# B&R Automation Studio project TD52 (part 119)

#### Cyclic.st - Cyclic code
```iecst
(*******************************************************************************
Ansl configuration for the Plant Communication

This code is confidential and proprietary to the INNIO Company.
It may not be used in any form, or reproduced in any manner, without the express
written permission of the INNIO Company.
Copyright, INNIO Company, 2024

Customized modifications: -
------------------------

History:
-------
V4.14.0	26.11.2024	Astner	Created Task

Instructions for use:
--------------------
The Configuration of the ANSL Communication is executed automatically when valid Parameter Values are configured.
If the Communication to the Master Control is redundant, set the variable bRedundantMasterEnabled in the Init Task.

Outstandings:
------------

*******************************************************************************)

PROGRAM _CYCLIC

	(* Parameters and Configuration Status for customized module *)
	OUT_HA.bPlantComCfgOk 		:= MM2VIS.tPlantComm.bCfg_OK;
		(* Start ANSL Configuration when parameter is set *)
	IF (EDGEPOS(Para.tPlantComm.bActive)) THEN
		MM2VIS.tPlantComm.bCfg_Err := FALSE;
		MM2VIS.tPlantComm.bCfg_OK := FALSE;
		MM2VIS.tPlantComm.bCfg_Rst := FALSE;
		iSTEP := GET_MODULE_NR;
	(* Stop ANSL Communication when parameter is unset *)
	ELSIF (EDGENEG(Para.tPlantComm.bActive)) THEN
		iSTEP := STOP_ANSL_COM;
		(* Exit Programm if parameter is not set *)
	ELSIF (NOT Para.tPlantComm.bActive AND NOT bPlantCommStopInProgress) THEN
		RETURN;
	END_IF;

	CASE iSTEP OF
		DATAOBJ_ERROR:
			(* Set HMI Diagnostics Error *)
			MM2VIS.tPlantComm.bCfg_Err := TRUE;
			MM2VIS.tPlantComm.bCfg_OK := FALSE;
			MM2VIS.tPlantComm.bCfg_Rst := FALSE;
			RETURN;
		ANSL_ERROR:
			(* Set HMI Diagnostics Error *)
			MM2VIS.tPlantComm.bCfg_Err := TRUE;
			MM2VIS.tPlantComm.bCfg_OK := FALSE;
			MM2VIS.tPlantComm.bCfg_Rst := FALSE;
			RETURN;
		GET_MODULE_NR:
			(* Set Engine Number to 1 for WinMOD Simulation *)
			IF (OUT_HA.bSimWinMOD_Active) THEN
				iThisEngineNr := 1;
				itoa(iThisEngineNr, ADR(strThisEngineNr));
				(* Reset Error bits*)
				MM2VIS.tPlantComm.bCfg_Err := FALSE;
				MM2VIS.tPlantComm.bCfg_OK := FALSE;
				MM2VIS.tPlantComm.bCfg_Rst := FALSE;
				(* Go to the next step *)
				iSTEP := PREP_DATAOBJ;
				RETURN;
			END_IF;
			(* Use Engine Number from HMI *)
			IF (IN_HA.iModule >= 1 AND IN_HA.iModule <= 32) THEN
				iThisEngineNr := IN_HA.iModule;
				itoa(iThisEngineNr, ADR(strThisEngineNr));
			ELSE
				MM2VIS.tPlantComm.bCfg_Err := TRUE;
				MM2VIS.tPlantComm.bCfg_OK := FALSE;
				MM2VIS.tPlantComm.bCfg_Rst := FALSE;
				RETURN;
			END_IF;
			IF (Para.tPlantComm.iEng_Num_Min = 0 AND Para.tPlantComm.iEng_Num_Max = 0) THEN
				bEng2EngComEnabled := FALSE;
			ELSIF (Para.tPlantComm.iEng_Num_Min > Para.tPlantComm.iEng_Num_Max) THEN
				MM2VIS.tPlantComm.bCfg_Err := TRUE;
				MM2VIS.tPlantComm.bCfg_OK := FALSE;
				MM2VIS.tPlantComm.bCfg_Rst := FALSE;
				RETURN;
			(* Out of bounds check *)
			ELSIF (Para.tPlantComm.iEng_Num_Min < 1 OR Para.tPlantComm.iEng_Num_Min > 32 OR Para.tPlantComm.iEng_Num_Max < 1 OR Para.tPlantComm.iEng_Num_Max > 32) THEN
				MM2VIS.tPlantComm.bCfg_Err := TRUE;
				MM2VIS.tPlantComm.bCfg_OK := FALSE;
				MM2VIS.tPlantComm.bCfg_Rst := FALSE;
				RETURN;
			ELSE
				bEng2EngComEnabled := TRUE;
				iEngNumMin := Para.tPlantComm.iEng_Num_Min;
				iEngNumMax := Para.tPlantComm.iEng_Num_Max;
			END_IF;
			IF (Para.tPlantComm.iMas_Num_Min = 0 AND Para.tPlantComm.iMas_Num_Max = 0) THEN
				bEng2MasComEnabled := FALSE;
			ELSIF (Para.tPlantComm.iMas_Num_Min > Para.tPlantComm.iMas_Num_Max) THEN
				MM2VIS.tPlantComm.bCfg_Err := TRUE;
				MM2VIS.tPlantComm.bCfg_OK := FALSE;
				MM2VIS.tPlantComm.bCfg_Rst := FALSE;
				RETURN;
			ELSE
				bEng2MasComEnabled := TRUE;
				iMasNumMin := Para.tPlantComm.iMas_Num_Min;
				iMasNumMax := Para.tPlantComm.iMas_Num_Max;
			END_IF;

			(* Reset Error bits and continue with the next step *)
			MM2VIS.tPlantComm.bCfg_Err := FALSE;
			MM2VIS.tPlantComm.bCfg_OK := FALSE;
			MM2VIS.tPlantComm.bCfg_Rst := FALSE;
			iSTEP := PREP_DATAOBJ;

		PREP_DATAOBJ:
			(*** Creation of the ANSL Configuration Data Object ***)

			(* ANSL Header *)
			strcat(pANSL_config, ADR('<?xml version ="1.0" encoding="utf-8"?>'));
			strcat(pANSL_config, ADR('<AnslClient>'));
			strcat(pANSL_config, ADR('<Diag TimeStamp="HalIO::tDiagClient.TimeStamp" ClientConn="HalIO::tDiagClient.Conn" ClientConnErr="HalIO::tDiagClient.ConnErr"/>'));

			(********************************************************************)
			(*																	*)
			(*                   Communication to Master						*)
			(*																	*)
			(********************************************************************)

			IF (bEng2MasComEnabled) THEN
				IF (NOT bRedundantMasterEnabled) THEN
					(* Add configured Masters to communication *)
					FOR x:=iMasNumMin TO iMasNumMax DO
						(* Check length of config object *)
						IF strlen(pANSL_config) > iANSL_config_length_max - 1000 THEN
							iSTEP := DATAOBJ_ERROR;
							RETURN;
						END_IF;
						(* Convert current asset numbers to strings *)
						strCurrentAssetNum 	:= '';
						strCurrentAssetSub 	:= '';
						strCurrentAssetIP 	:= '';
						itoa(x, ADR(strCurrentAssetNum));
						itoa(iMastersSUB[x], ADR(strCurrentAssetSub));
						itoa(iMastersIP[x], ADR(strCurrentAssetIP));

						//Line 1
						strcat(pANSL_config, ADR('<Connection ConnName="Master'));
						strcat(pANSL_config, ADR(strCurrentAssetNum));
						strcat(pANSL_config, ADR('" TargetAddr="192.168.'));
						strcat(pANSL_config, ADR(strCurrentAssetSub));
						strcat(pANSL_config, ADR('.'));
						strcat(pANSL_config, ADR(strCurrentAssetIP));
						strcat(pANSL_config, ADR('" AnslPort="11179" Timeout="5000" SendDelay="2" BfSize="65536" ConnMode="0" EnableSSL="1" SSLConfig="SSL_Eng'));
						strcat(pANSL_config, ADR(strThisEngineNr));
						strcat(pANSL_config, ADR('" PW="'));
						strcat(pANSL_config, ADR(strAnsl_Com_Pw));
						strcat(pANSL_config, ADR('">'));
						// Line 2
						strcat(pANSL_config, ADR('<Diag ConnErr="HalIO::tDiagMaster['));
						strcat(pANSL_config, ADR(strCurrentAssetNum));
						strcat(pANSL_config, ADR('].Err" ConnPvWrite="HalIO::tDiagMaster['));
						strcat(pANSL_config, ADR(strCurrentAssetNum));
						strcat(pANSL_config, ADR('].PvWrite" ConnPvWriteErr="HalIO::tDiagMaster['));
						strcat(pANSL_config, ADR(strCurrentAssetNum));
						strcat(pANSL_config, ADR('].PvWriteErr" ConnPvReadErr="HalIO::tDiagMaster['));
						strcat(pANSL_config, ADR(strCurrentAssetNum));
						strcat(pANSL_config, ADR('].PvReadErr"/>'));
						// Line 3
						strcat(pANSL_config, ADR('<PVS>'));
						// Line 4
						strcat(pANSL_config, ADR('<Read LocalPvName="HalIO::tPlantCom_M2E_In_100ms['));
						strcat(pANSL_config, ADR(strCurrentAssetNum));
						strcat(pANSL_config, ADR(']" RemotePvName="HalIO::tPlantCom_M2E_Out_100ms['));
						strcat(pANSL_config, ADR(strThisEngineNr));
						strcat(pANSL_config, ADR(']" DefaultValue="0" SyncPv="0" RefreshRate="100" Hysteresis="0"/>'));
						// Line 5
						strcat(pANSL_config, ADR('<Read LocalPvName="HalIO::tPlantCom_M2E_In_10ms['));
						strcat(pANSL_config, ADR(strCurrentAssetNum));
						strcat(pANSL_config, ADR(']" RemotePvName="HalIO::tPlantCom_M2E_Out_10ms['));
						strcat(pANSL_config, ADR(strThisEngineNr));
						strcat(pANSL_config, ADR(']" DefaultValue="0" SyncPv="0" RefreshRate="10" Hysteresis="0"/>'));
						// Line 6
						strcat(pANSL_config, ADR('</PVS>'));
						// Line 7
						strcat(pANSL_config, ADR('</Connection>'));
					END_FOR
				ELSE
					(********************************************************************)
					(*																	*)
					(*                 Communication to Redundant Master				*)
					(*																	*)
					(********************************************************************)

					(* Check length of config object *)
					IF strlen(pANSL_config) > iANSL_config_length_max - 1000 THEN
						iSTEP := DATAOBJ_ERROR;
						RETURN;
					END_IF;
					(* Convert current asset numbers to strings *)
					strCurrentAssetNum 	:= '';
					strCurrentAssetSub 	:= '';
					strCurrentAssetIP 	:= '';
					itoa(1, ADR(strCurrentAssetNum));
					itoa(iMastersSUB[1], ADR(strCurrentAssetSub));
					itoa(iMastersIP[1], ADR(strCurrentAssetIP));

					//Line 1
					strcat(pANSL_config, ADR('<Connection ConnName="Master'));
					strcat(pANSL_config, ADR(strCurrentAssetNum));
					strcat(pANSL_config, ADR('" TargetAddr="192.168.'));
					strcat(pANSL_config, ADR(strCurrentAssetSub));
					strcat(pANSL_config, ADR('.'));
					strcat(pANSL_config, ADR(strCurrentAssetIP));
					strcat(pANSL_config, ADR('" AnslPort="11169" Timeout="5000" SendDelay="2" BfSize="65536" ConnMode="1" EnableSSL="0" SSLConfig="SSL_Eng'));
					strcat(pANSL_config, ADR(strThisEngineNr));
					strcat(pANSL_config, ADR('" PW="'));
					strcat(pANSL_config, ADR(strAnsl_Com_Pw));
					strcat(pANSL_config, ADR('">'));
					// Line 2
					strcat(pANSL_config, ADR('<Diag ConnErr="HalIO::tDiagMaster['));
					strcat(pANSL_config, ADR(strCurrentAssetNum));
					strcat(pANSL_config, ADR('].Err" ConnPvWrite="HalIO::tDiagMaster['));
					strcat(pANSL_config, ADR(strCurrentAssetNum));
					strcat(pANSL_config, ADR('].PvWrite" ConnPvWriteErr="HalIO::tDiagMaster['));
					strcat(pANSL_config, ADR(strCurrentAssetNum));
					strcat(pANSL_config, ADR('].PvWriteErr" ConnPvReadErr="HalIO::tDiagMaster['));
					strcat(pANSL_config, ADR(strCurrentAssetNum));
					strcat(pANSL_config, ADR('].PvReadErr" RedConnActIpAddr="HalIO::tDiagMaster['));
					strcat(pANSL_config, ADR(strCurrentAssetNum));
					strcat(pANSL_config, ADR('].RedConnActIpAddr" RedConnAct="HalIO::tDiagMaster['));
					strcat(pANSL_config, ADR(strCurrentAssetNum));
					strcat(pANSL_config, ADR('].RedConnAct" RedConnState="HalIO::tDiagMaster['));
					strcat(pANSL_config, ADR(strCurrentAssetNum));
					strcat(pANSL_config, ADR('].RedConnState"/>'));
					// Line 3
					strcat(pANSL_config, ADR('<PVS>'));
					// Line 4
					strcat(pANSL_config, ADR('<Read LocalPvName="HalIO::tPlantCom_M2E_In_100ms['));
					strcat(pANSL_config, ADR(strCurrentAssetNum));
					strcat(pANSL_config, ADR(']" RemotePvName="HalIO::tPlantCom_M2E_Out_100ms['));
					strcat(pANSL_config, ADR(strThisEngineNr));
					strcat(pANSL_config, ADR(']" DefaultValue="0" SyncPv="0" RefreshRate="100" Hysteresis="0"/>'));
					// Line 5
					strcat(pANSL_config, ADR('<Read LocalPvName="HalIO::tPlantCom_M2E_In_10ms['));
					strcat(pANSL_config, ADR(strCurrentAssetNum));
					strcat(pANSL_config, ADR(']" RemotePvName="HalIO::tPlantCom_M2E_Out_10ms['));
					strcat(pANSL_config, ADR(strThisEngineNr));
					strcat(pANSL_config, ADR(']" DefaultValue="0" SyncPv="0" RefreshRate="10" Hysteresis="0"/>'));
					// Line 6
					strcat(pANSL_config, ADR('</PVS>'));
					// Line 7
					strcat(pANSL_config, ADR('</Connection>'));
				END_IF
			END_IF

			(********************************************************************)
			(*																	*)
			(*                   Communication to Engines						*)
			(*																	*)
			(********************************************************************)

			IF (bEng2EngComEnabled) THEN
				(* Add configured Engines to communication *)
				FOR x:=iEngNumMin TO iEngNumMax DO
					(* Check length of config object *)
					IF strlen(pANSL_config) > iANSL_config_length_max - 1000 THEN
						iSTEP := DATAOBJ_ERROR;
						RETURN;
					END_IF;

					IF (x <> iThisEngineNr) THEN
						(* Convert current asset numbers to strings *)
						strCurrentAssetNum 	:= '';
						strCurrentAssetSub 	:= '';
						strCurrentAssetIP 	:= '';
						itoa(x, ADR(strCurrentAssetNum));
						itoa(iEnginesSUB[x], ADR(strCurrentAssetSub));
						itoa(iEnginesIP[x], ADR(strCurrentAssetIP));

						//Line 1
						strcat(pANSL_config, ADR('<Connection ConnName="Engine'));
						strcat(pANSL_config, ADR(strCurrentAssetNum));
						strcat(pANSL_config, ADR('" TargetAddr="192.168.'));
						strcat(pANSL_config, ADR(strCurrentAssetSub));
						strcat(pANSL_config, ADR('.'));
						strcat(pANSL_config, ADR(strCurrentAssetIP));
						strcat(pANSL_config, ADR('" AnslPort="11179" Timeout="5000" SendDelay="2" BfSize="65536" ConnMode="0" EnableSSL="1" SSLConfig="SSL_Eng'));
						strcat(pANSL_config, ADR(strThisEngineNr));
						strcat(pANSL_config, ADR('"> PW="'));
						strcat(pANSL_config, ADR(strAnsl_Com_Pw));
						strcat(pANSL_config, ADR('"'));

						// Line 2
						strcat(pANSL_config, ADR('<Diag ConnErr="HalIO::tDiagEngine['));
						strcat(pANSL_config, ADR(strCurrentAssetNum));
						strcat(pANSL_config, ADR('].Err" ConnPvWrite="HalIO::tDiagEngine['));
						strcat(pANSL_config, ADR(strCurrentAssetNum));
						strcat(pANSL_config, ADR('].PvWrite" ConnPvWriteErr="HalIO::tDiagEngine['));
						strcat(pANSL_config, ADR(strCurrentAssetNum));
						strcat(pANSL_config, ADR('].PvWriteErr" ConnPvReadErr="HalIO::tDiagEngine['));
						strcat(pANSL_config, ADR(strCurrentAssetNum));
						strcat(pANSL_config, ADR('].PvReadErr"/>'));
						// Line 3
						strcat(pANSL_config, ADR('<PVS>'));
						// Line 4
						strcat(pANSL_config, ADR('<Read LocalPvName="HalIO::tPlantCom_E2E_In_100ms['));
						strcat(pANSL_config, ADR(strCurrentAssetNum));
						strcat(pANSL_config, ADR(']" RemotePvName="HalIO::tPlantCom_E2E_Out_100ms" DefaultValue="0" SyncPv="0" RefreshRate="100" Hysteresis="0"/>'));
						// Line 5
						strcat(pANSL_config, ADR('<Read LocalPvName="HalIO::tPlantCom_E2E_In_10ms['));
						strcat(pANSL_config, ADR(strCurrentAssetNum));
						strcat(pANSL_config, ADR(']" RemotePvName="HalIO::tPlantCom_E2E_Out_10ms" DefaultValue="0" SyncPv="0" RefreshRate="10" Hysteresis="0"/>'));
						// Line 6
						strcat(pANSL_config, ADR('</PVS>'));
						// Line 7
						strcat(pANSL_config, ADR('</Connection>'));
					END_IF
				END_FOR
			END_IF

			(* ANSL Footer*)
			strcat(pANSL_config, ADR('</AnslClient>'));

			(* Reset Error bits and continue with the next step *)
			MM2VIS.tPlantComm.bCfg_Err 				:= FALSE;
			MM2VIS.tPlantComm.bCfg_OK 				:= FALSE;
			MM2VIS.tPlantComm.bCfg_Rst 				:= FALSE;
			iSTEP := PREP_CHECK_DATAOBJ_STATUS;
		PREP_CHECK_DATAOBJ_STATUS:
			(* Prepare DataObjInfo Function Block *)
			xDatObjInfo_Ansl_Cfg.enable 			:= TRUE;
			xDatObjInfo_Ansl_Cfg.pName 				:= ADR(strAnslDataObjName);
			iSTEP := CHECK_DATAOBJ_STATUS;
		CHECK_DATAOBJ_STATUS:
			(* Check if DataObj already exists or has another error *)
			xDatObjInfo_Ansl_Cfg();
			(* Data object already exists *)
			IF (xDatObjInfo_Ansl_Cfg.status = ERR_OK) THEN
				xDatObjDelete_Ansl_Cfg.enable 		:= TRUE;
				xDatObjDelete_Ansl_Cfg.ident 		:= xDatObjInfo_Ansl_Cfg.ident;
				iSTEP := DELETE_DATAOBJ;
			ELSIF (xDatObjInfo_Ansl_Cfg.status = doERR_MODULNOTFOUND) THEN
				xDatObjCreate_Ansl_Cfg.enable 		:= TRUE;
				xDatObjCreate_Ansl_Cfg.pName 		:= ADR(strAnslDataObjName);
				xDatObjCreate_Ansl_Cfg.pCpyData 	:= pANSL_config;
				xDatObjCreate_Ansl_Cfg.MemType 		:= doUSRROM;
				xDatObjCreate_Ansl_Cfg.len 			:= strlen(pANSL_config);
				iSTEP 								:= CREATE_DATAOBJ;
			ELSIF (xDatObjInfo_Ansl_Cfg.status <> ERR_FUB_BUSY) THEN
				iSTEP 							:= DATAOBJ_ERROR;
			END_IF;
		DELETE_DATAOBJ:
			(* Delete Dataobj *)
			xDatObjDelete_Ansl_Cfg();
			IF (xDatObjDelete_Ansl_Cfg.status = ERR_OK) THEN
				xDatObjCreate_Ansl_Cfg.enable		:= TRUE;
				iSTEP 								:= CREATE_DATAOBJ;
			ELSIF (xDatObjDelete_Ansl_Cfg.status <> ERR_FUB_BUSY) THEN
				iSTEP						 		:= DATAOBJ_ERROR;
			END_IF;
		CREATE_DATAOBJ:
			IF (xDatObjCreate_Ansl_Cfg.len = 0) THEN
				iSTEP := PREP_DATAOBJ;
				RETURN;
			END_IF
			xDatObjCreate_Ansl_Cfg();
			IF (xDatObjCreate_Ansl_Cfg.status = ERR_OK) THEN
				strANSL_config 					:= '';
				xANSLClientStart.enable 		:= TRUE;
				xANSLClientStart.dataObjName 	:= strAnslDataObjName;
				iSTEP 							:= START_ANSL_COM;
			ELSIF (xDatObjCreate_Ansl_Cfg.status <> ERR_FUB_BUSY) THEN
				iSTEP						 	:= DATAOBJ_ERROR;
			END_IF;
		START_ANSL_COM:
			(* Only start ANSL Communication after all Software modules are loaded and running *)
			xANSLClientStart();
			IF (xANSLClientStart.status = ERR_OK) THEN
				xDatObjCreate_Ansl_Cfg.enable := FALSE;
				xDatObjDelete_Ansl_Cfg.enable := FALSE;
				xDatObjInfo_Ansl_Cfg.enable 	:= FALSE;
				MM2VIS.tPlantComm.bCfg_OK 	:= TRUE;
				iSTEP := PREP_ANSL_DIAGNOSTICS;
			ELSIF (xANSLClientStart.status <> ERR_FUB_BUSY) THEN
				iSTEP 						:= ANSL_ERROR;
			END_IF
		STOP_ANSL_COM:
			// todo test behaviour
			bPlantCommStopInProgress 			:= TRUE;
			xANSLClientStop.enable 				:= TRUE;
			xANSLClientStop.dataObjName 		:= strAnslDataObjName;
			xANSLClientStop();
			IF (xANSLClientStop.status = ERR_OK OR xANSLClientStop.status = asANSL_ERR_CLIENT_NOT_EXIST) THEN
				MM2VIS.tPlantComm.bCfg_OK 		:= FALSE;
				bPlantCommStopInProgress 		:= FALSE;
				(* Reset FUBs *)
				xANSLClientStart.dataObjName 	:= '';
				xANSLClientStart.enable			:= FALSE;
				xDatObjCreate_Ansl_Cfg.enable	:= FALSE;
				xDatObjCreate_Ansl_Cfg.len		:= 0;
				xDatObjCreate_Ansl_Cfg.pCpyData	:= 0;
				xDatObjInfo_Ansl_Cfg.enable		:= FALSE;
				xDatObjInfo_Ansl_Cfg.pName		:= 0;
				xDatObjDelete_Ansl_Cfg.enable	:= FALSE;
				xDatObjDelete_Ansl_Cfg.ident	:= 0;
				iSTEP := GET_MODULE_NR;
			ELSIF (xANSLClientStop.status <> ERR_FUB_BUSY) THEN
				iSTEP 							:= ANSL_ERROR;
			END_IF;
		PREP_ANSL_DIAGNOSTICS:
			iSTEP := ANSL_DIAGNOSTICS;
		ANSL_DIAGNOSTICS:
			(* Check for configuration changes *)
			IF (iEngNumMin <> Para.tPlantComm.iEng_Num_Min OR
				iEngNumMax <> Para.tPlantComm.iEng_Num_Max OR
				iMasNumMin <> Para.tPlantComm.iMas_Num_Min OR
				iMasNumMax <> Para.tPlantComm.iMas_Num_Max) THEN
				iSTEP := STOP_ANSL_COM;
			END_IF
			(* Evaluate Masters *)
			iNum_InterruptedMasters := 0;
			FOR x:=iMasNumMin TO iMasNumMax DO
				MM2VIS.tPlantComm.bMas_Ena[x] := tDiagMaster[x].Err = 0 AND tDiagMaster[x].PvReadErr = 0;
				IF (tDiagMaster[x].Err <> 0 OR tDiagMaster[x].PvReadErr <> 0) THEN
					iNum_InterruptedMasters := iNum_InterruptedMasters + 1;
				END_IF
			END_FOR

			(* Evaluate Engines *)
			iNum_InterruptedEngines := 0;
			FOR x:=iEngNumMin TO iEngNumMax DO
				IF (x = iThisEngineNr) THEN
					MM2VIS.tPlantComm.bEng_Ena[x] := TRUE;
				ELSE
					MM2VIS.tPlantComm.bEng_Ena[x] := tDiagEngine[x].Err = 0 AND tDiagEngine[x].PvReadErr = 0 AND x <> iThisEngineNr;
					IF (tDiagEngine[x].Err <> 0 OR tDiagEngine[x].PvReadErr <> 0) THEN
						iNum_InterruptedEngines := iNum_InterruptedEngines + 1;
					END_IF
				END_IF
			END_FOR

			(* Set warning variable *)
			bPlantComm_interrupted := iNum_InterruptedEngines <> 0 OR iNum_InterruptedMasters <> 0;

			(* Set/Unset GoodQual Values on connection interuptions/establishment *)
			FOR x:= iEngNumMin TO iEngNumMax DO
				IF (EDGENEG(MM2VIS.tPlantComm.bEng_Ena[x])) THEN
					FOR idx:=0 TO iDigArrayMax100ms DO
						tPlantCom_E2E_In_100ms[x].digitalSignals[idx].GoodQual := FALSE;
					END_FOR
					FOR idx:=0 TO iDigArrayMax10ms DO
						tPlantCom_E2E_In_10ms[x].digitalSignals[idx].GoodQual := FALSE;
					END_FOR
					FOR idx:=0 TO iAnaArrayMax100ms DO
						tPlantCom_E2E_In_100ms[x].analogSignals[idx].GoodQual := FALSE;
					END_FOR
					FOR idx:=0 TO iAnaArrayMax10ms DO
						tPlantCom_E2E_In_10ms[x].analogSignals[idx].GoodQual := FALSE;
					END_FOR
				END_IF
			END_FOR
			FOR x:= iMasNumMin TO iMasNumMax DO
				IF (EDGENEG(MM2VIS.tPlantComm.bMas_Ena[x])) THEN
					FOR idx:=0 TO iDigArrayMax100ms DO
						tPlantCom_M2E_In_100ms[x].digitalSignals[idx].GoodQual := FALSE;
					END_FOR
					FOR idx:=0 TO iDigArrayMax10ms DO
						tPlantCom_M2E_In_10ms[x].digitalSignals[idx].GoodQual := FALSE;
					END_FOR
					FOR idx:=0 TO iAnaArrayMax100ms DO
						tPlantCom_M2E_In_100ms[x].analogSignals[idx].GoodQual := FALSE;
					END_FOR
					FOR idx:=0 TO iAnaArrayMax10ms DO
						tPlantCom_M2E_In_10ms[x].analogSignals[idx].GoodQual := FALSE;
					END_FOR
				END_IF
			END_FOR
	END_CASE
END_PROGRAM
```

#### Init.st - Init code
```iecst
(*******************************************************************************
Ansl configuration for the Plant Communication

This code is confidential and proprietary to the INNIO Company.
It may not be used in any form, or reproduced in any manner, without the express
written permission of the INNIO Company.
Copyright, INNIO Company, 2024

Customized modifications: -
------------------------

History:
-------
V4.14.0	26.11.2024	Astner	Created Task

Instructions for use:
--------------------
The Configuration of the ANSL Communication is executed automatically when valid Parameter Values are configured.
If the Communication to the Master Control is redundant, set the variable bRedundantMasterEnabled in the Init Task.

Outstandings:
------------

*******************************************************************************)

PROGRAM _INIT
	(* Master 1 is redundant *)
	bRedundantMasterEnabled := FALSE;

	(* Default diagnostic bits *)
	MM2VIS.tPlantComm.bCfg_Err := FALSE;
	MM2VIS.tPlantComm.bCfg_OK  := FALSE;
	MM2VIS.tPlantComm.bCfg_Rst := FALSE;

	(* IP & SUBNET Masks *)
	FOR x:=1 TO 4 DO
		iMastersSUB[x]	:=	122;
		iMastersIP[x] 	:= 	30 + x;
	END_FOR

	FOR x:=1 TO 32 DO
		iEnginesSUB[x]	:=	122;
		iEnginesIP[x] 	:= 	10 + x;
	END_FOR
	(* Initialize Configuration Strings and Pointers *)
	strAnslDataObjName := 'HalIO::ANSLCom';
	strThisEngineNr := '';
	strCurrentAssetIP := '';
	strCurrentAssetSub := '';
	strCurrentAssetNum := '';
	strANSL_config := '';
	pANSL_config := ADR(strANSL_config);
	strAnsl_Com_Pw := 'vvsZKl2WtfuUhIlKaiANBLBnqHMr7jLXo7MDs/K0/P5wtUylYnR+0YUUjcfS9T0G';

	iSTEP := GET_MODULE_NR;

	tDiagClient;
	tDiagMaster;
	tDiagEngine;

END_PROGRAM
```

#### Variables.var - Local variables
```iecst
(*Configuration Step Variables*)
VAR
	iSTEP : USINT := 0;
END_VAR
VAR CONSTANT
	DATAOBJ_ERROR : USINT := 0;
	ANSL_ERROR : USINT := 1;
	GET_MODULE_NR : USINT := 2;
	PREP_DATAOBJ : USINT := 3;
	PREP_CHECK_DATAOBJ_STATUS : USINT := 4;
	CHECK_DATAOBJ_STATUS : USINT := 5;
	DELETE_DATAOBJ : USINT := 6;
	CREATE_DATAOBJ : USINT := 7;
	START_ANSL_COM : USINT := 8;
	STOP_ANSL_COM : USINT := 9;
	PREP_ANSL_DIAGNOSTICS : USINT := 10;
	ANSL_DIAGNOSTICS : USINT := 11;
END_VAR
VAR
	bPlantCommStopInProgress : BOOL := FALSE;
END_VAR
(*ANSL Config Variables*)
VAR
	strAnsl_Com_Pw : STRING[64] := ''; (*Password Hash for the encrypted ANSL Communication*)
	iThisEngineNr : USINT := 0; (*Engine number of this Engine*)
	strThisEngineNr : STRING[16] := ''; (*Engine number of this Engine*)
	iMastersSUB : ARRAY[0..4] OF USINT; (*Subnet Part of the IP of each master*)
	iMastersIP : ARRAY[0..4] OF USINT; (*Host Part of the IP of each master*)
	iEnginesSUB : ARRAY[0..32] OF USINT; (*Subnet Part of the IP of each engine*)
	iEnginesIP : ARRAY[0..32] OF USINT; (*Host Part of the IP of each engine*)
	idx : USINT := 0; (*loop iterator used to iterate over signals*)
	x : USINT := 0; (*loop iterator used to iterate over the communication participants*)
END_VAR
VAR CONSTANT
	iANSL_config_length_max : UINT := 60000; (*max dataobject length*)
END_VAR
VAR
	strANSL_config : STRING[iANSL_config_length_max] := ''; (*Ansl configuration string*)
	pANSL_config : UDINT := 0; (*Pointer to the Ansl configuration string*)
	strCurrentAssetNum : STRING[16] := ''; (*Strings of the dynamic values that are used to build the ansl dataoject*)
	strCurrentAssetSub : STRING[16] := ''; (*Strings of the dynamic values that are used to build the ansl dataoject*)
	strCurrentAssetIP : STRING[16] := ''; (*Strings of the dynamic values that are used to build the ansl dataoject*)
END_VAR
(*ANSL Dataobject Variables*)
VAR
	xDatObjInfo_Ansl_Cfg : DatObjInfo := (0);
	xDatObjDelete_Ansl_Cfg : DatObjDelete := (0);
	xDatObjCreate_Ansl_Cfg : DatObjCreate := (0);
	strAnslDataObjName : STRING[32] := '';
END_VAR
(*ANSL Communication FUBs*)
VAR
	xANSLClientStart : AsANSLClientStart := (0);
	xANSLClientStop : AsANSLClientStop := (0);
END_VAR
```

### Program Logical/HalIO/PlantCommunication/XComHmi (IEC, version 4.14.0)

#### Cyclic.st - Cyclic code
```iecst
(*******************************************************************************
Hmi Logic for the Plant Communication Diagnostics and Forcing screen

This code is confidential and proprietary to the INNIO Company.
It may not be used in any form, or reproduced in any manner, without the express
written permission of the INNIO Company.
Copyright, INNIO Company, 2024

Customized modifications: -
------------------------

History:
-------
V4.14.0	26.11.2024	Astner	Created Task

Instructions for use: -
--------------------

Outstandings:
------------

*******************************************************************************)
PROGRAM _CYCLIC

	IF (NOT Para.tPlantComm.bActive) THEN
		FOR x := 1 TO 4 DO
			MM2VIS.tPlantComm.bMas_Ena[x] := FALSE;
		END_FOR
		FOR x := 1 TO 32 DO
			MM2VIS.tPlantComm.bEng_Ena[x] := FALSE;
		END_FOR
	END_IF;

	(* Exit if configuration fails or not active *)
	IF (NOT MM2VIS.tPlantComm.bCfg_OK OR NOT Para.tPlantComm.bActive) THEN
		RETURN;
	END_IF;

	IF (Para.tPlantComm.iEng_Num_Min > Para.tPlantComm.iEng_Num_Max) THEN
		Para.tPlantComm.iEng_Num_Max := Para.tPlantComm.iEng_Num_Min;
	END_IF;
	IF (Para.tPlantComm.iMas_Num_Min > Para.tPlantComm.iMas_Num_Max) THEN
		Para.tPlantComm.iMas_Num_Max := Para.tPlantComm.iMas_Num_Min;
	END_IF;
	iEngNumMin := Para.tPlantComm.iEng_Num_Min;
	iEngNumMax := Para.tPlantComm.iEng_Num_Max;
	iMasNumMin := Para.tPlantComm.iMas_Num_Min;
	iMasNumMax := Para.tPlantComm.iMas_Num_Max;

	(**********************************************************)
	(*      			HMI Diagnostics					      *)
	(**********************************************************)

	tHmiDiag.bSelectionChange := FALSE;

	(*Signal Type changed in the Diagnostic screen selection *)
	IF (VIS2MM.tPlantComm.iIO_Typ <> tHmiDiag.iIO_Typ) THEN
		(* Set the IO Type: AI, DI, AO, DO *)
		tHmiDiag.iIO_Typ := VIS2MM.tPlantComm.iIO_Typ;

		(* Reset the direction selection on the HMI *)
		VIS2MM.tPlantComm.iIO_Typ_Dir := NO_SELECTION;
		VIS2MM.tPlantComm.iIO_Typ_Dir_Num := NO_SELECTION;
		VIS2MM.tPlantComm.iNum_Start := 0;
		tHmiDiag.iIO_Typ_Dir := NO_SELECTION;
		tHmiDiag.iIO_Typ_Dir_Num := NO_SELECTION;
		tHmiDiag.iStartIdx := NO_SELECTION;

		tHmiDiag.bSelectionChange := TRUE;
	END_IF;

	(* Signal Direction changed in the Diagnostic screen selection *)
	IF (VIS2MM.tPlantComm.iIO_Typ_Dir <> tHmiDiag.iIO_Typ_Dir) THEN
		(* Set the Signal Direction: FROM Master/Engine TO Master/Engine *)
		IF (tHmiDiag.iIO_Typ = PlantComm_AI OR tHmiDiag.iIO_Typ = PlantComm_DI) THEN // Input only allows Signals FROM Master/Engine
			IF (VIS2MM.tPlantComm.iIO_Typ_Dir = FROM_MASTER OR VIS2MM.tPlantComm.iIO_Typ_Dir = FROM_ENGINE) THEN
				tHmiDiag.iIO_Typ_Dir := VIS2MM.tPlantComm.iIO_Typ_Dir;
			ELSE
				NO_SELECTION;
				tHmiDiag.iIO_Typ_Dir := NO_SELECTION;
				VIS2MM.tPlantComm.iIO_Typ_Dir := NO_SELECTION;
			END_IF
		ELSIF (tHmiDiag.iIO_Typ = PlantComm_AO OR tHmiDiag.iIO_Typ = PlantComm_DO) THEN // Output only allows Signals TO Master/Engine
			IF (VIS2MM.tPlantComm.iIO_Typ_Dir = TO_MASTER OR VIS2MM.tPlantComm.iIO_Typ_Dir = TO_ENGINE) THEN
				tHmiDiag.iIO_Typ_Dir := VIS2MM.tPlantComm.iIO_Typ_Dir;
			ELSE
				NO_SELECTION;
				tHmiDiag.iIO_Typ_Dir := NO_SELECTION;
				VIS2MM.tPlantComm.iIO_Typ_Dir := NO_SELECTION;
			END_IF
		ELSE
			VIS2MM.tPlantComm.iIO_Typ_Dir := tHmiDiag.iIO_Typ_Dir;
		END_IF;
		(* Set the Dir_Num limits *)
		IF (VIS2MM.tPlantComm.iIO_Typ_Dir = FROM_MASTER OR VIS2MM.tPlantComm.iIO_Typ_Dir = TO_MASTER) THEN
			MM2VIS.tPlantComm.iIO_Typ_Dir_Num_Max := iMasNumMax;
			MM2VIS.tPlantComm.iIO_Typ_Dir_Num_Min := iMasNumMin;
			VIS2MM.tPlantComm.iIO_Typ_Dir_Num	  := iMasNumMin;
		ELSIF (VIS2MM.tPlantComm.iIO_Typ_Dir = FROM_ENGINE OR VIS2MM.tPlantComm.iIO_Typ_Dir = TO_ENGINE) THEN
			MM2VIS.tPlantComm.iIO_Typ_Dir_Num_Max := iEngNumMax;
			MM2VIS.tPlantComm.iIO_Typ_Dir_Num_Min := iEngNumMin;
			VIS2MM.tPlantComm.iIO_Typ_Dir_Num	  := iEngNumMin;
		END_IF
		(* Reset the Asset Selection *)
		VIS2MM.tPlantComm.iNum_Start := NO_SELECTION;
		VIS2MM.tPlantComm.bFrc_Act := FALSE;
		VIS2MM.tPlantComm.bFrc_Gbl := FALSE;
		tHmiDiag.iIO_Typ_Dir_Num := VIS2MM.tPlantComm.iIO_Typ_Dir_Num;
		tHmiDiag.iStartIdx := NO_SELECTION;
		tHmiDiag.bSelectionChange := TRUE;
	END_IF

	(* Dir_Num Selection changed*)
	IF (VIS2MM.tPlantComm.iIO_Typ_Dir_Num <> tHmiDiag.iIO_Typ_Dir_Num) THEN
		(* Set the asset selection *)
		IF (tHmiDiag.iIO_Typ_Dir = FROM_MASTER OR tHmiDiag.iIO_Typ_Dir = TO_MASTER) THEN
			IF (VIS2MM.tPlantComm.iIO_Typ_Dir_Num >= iMasNumMin AND VIS2MM.tPlantComm.iIO_Typ_Dir_Num <= iMasNumMax) THEN
				tHmiDiag.iIO_Typ_Dir_Num := VIS2MM.tPlantComm.iIO_Typ_Dir_Num;
				tHmiDiag.bSelectionChange := TRUE;
			ELSE
				VIS2MM.tPlantComm.iIO_Typ_Dir_Num := tHmiDiag.iIO_Typ_Dir_Num;
			END_IF
		ELSIF (tHmiDiag.iIO_Typ_Dir = FROM_ENGINE OR tHmiDiag.iIO_Typ_Dir = TO_ENGINE) THEN
			IF (VIS2MM.tPlantComm.iIO_Typ_Dir_Num >= iEngNumMin AND VIS2MM.tPlantComm.iIO_Typ_Dir_Num <= iEngNumMax) THEN
				tHmiDiag.iIO_Typ_Dir_Num := VIS2MM.tPlantComm.iIO_Typ_Dir_Num;
				tHmiDiag.bSelectionChange := TRUE;
			ELSE
				VIS2MM.tPlantComm.iIO_Typ_Dir_Num := tHmiDiag.iIO_Typ_Dir_Num;
			END_IF
		ELSE
			VIS2MM.tPlantComm.iIO_Typ_Dir_Num := tHmiDiag.iIO_Typ_Dir_Num;
		END_IF
		VIS2MM.tPlantComm.iNum_Start := NO_SELECTION;
		tHmiDiag.iStartIdx := NO_SELECTION;
	END_IF
	(* Start Index Changed *)
	IF (VIS2MM.tPlantComm.iNum_Start <> tHmiDiag.iStartIdx) THEN
		tHmiDiag.iStartIdx := VIS2MM.tPlantComm.iNum_Start;
		tHmiDiag.bSelectionChange := TRUE;
	END_IF

	(* Unforce all Asset *)
	IF (VIS2MM.tPlantComm.bFrc_Act) THEN
		(* Reset HMI Selection of Force Active *)
		FOR x:=0 TO tHmiDiag.iDiagTableSize-1 DO
			VIS2MM.tPlantComm.bFrc[x] := FALSE;
		END_FOR
		(* Unforce all of the selected Asset *)
		IF (tHmiDiag.iIO_Typ_Dir = FROM_MASTER OR tHmiDiag.iIO_Typ_Dir = TO_MASTER) THEN
			IF (tHmiDiag.iIO_Typ_Dir_Num >= 1 AND tHmiDiag.iIO_Typ_Dir_Num <= 4) THEN
				(* Unforce Analog Inputs/Outputs *)
				FOR x:=0 TO tHmiDiag.iAnaSigCntE2M - 1 DO
					tPlantCom_M2E_In_Hmi[tHmiDiag.iIO_Typ_Dir_Num].bAnaForceActive[x] := FALSE;
					tPlantCom_E2M_Out_Hmi[tHmiDiag.iIO_Typ_Dir_Num].bAnaForceActive[x] := FALSE;
				END_FOR
				(* Unforce Digital Inputs/Outputs *)
				FOR x:=0 TO tHmiDiag.iDigSigCntE2M - 1 DO
					tPlantCom_M2E_In_Hmi[tHmiDiag.iIO_Typ_Dir_Num].bDigForceActive[x] := FALSE;
					tPlantCom_E2M_Out_Hmi[tHmiDiag.iIO_Typ_Dir_Num].bDigForceActive[x] := FALSE;
				END_FOR
				(* Set counter for forced signals to zero*)
				tPlantCom_M2E_In_Hmi[tHmiDiag.iIO_Typ_Dir_Num].iNum_ForcedValues 	:= 0;
				tPlantCom_E2M_Out_Hmi[tHmiDiag.iIO_Typ_Dir_Num].iNum_ForcedValues  	:= 0;
			END_IF
		ELSIF (tHmiDiag.iIO_Typ_Dir = FROM_ENGINE) THEN
			IF (tHmiDiag.iIO_Typ_Dir_Num >= 1 AND tHmiDiag.iIO_Typ_Dir_Num <= 32) THEN
				(* Unforce Analog Inputs *)
				FOR x:=0 TO tHmiDiag.iAnaSigCntE2E - 1 DO
					tPlantCom_E2E_In_Hmi[tHmiDiag.iIO_Typ_Dir_Num].bAnaForceActive[x] := FALSE;
				END_FOR
				(* Unforce Digital Inputs *)
				FOR x:=0 TO tHmiDiag.iDigSigCntE2E - 1 DO
					tPlantCom_E2E_In_Hmi[tHmiDiag.iIO_Typ_Dir_Num].bDigForceActive[x] := FALSE;
				END_FOR
				tPlantCom_E2E_In_Hmi[tHmiDiag.iIO_Typ_Dir_Num].iNum_ForcedValues := 0;
			END_IF
		ELSIF (tHmiDiag.iIO_Typ_Dir = TO_ENGINE) THEN
			(* Unforce Analog Outputs *)
			FOR x:=0 TO tHmiDiag.iAnaSigCntE2E - 1 DO
				tPlantCom_E2E_Out_Hmi.bAnaForceActive[x] := FALSE;
			END_FOR
			(* Unforce Digital Outputs *)
			FOR x:=0 TO tHmiDiag.iDigSigCntE2E - 1 DO
				tPlantCom_E2E_Out_Hmi.bDigForceActive[x] := FALSE;
			END_FOR
			tPlantCom_E2E_Out_Hmi.iNum_ForcedValues	:= 0;
		END_IF
		VIS2MM.tPlantComm.bFrc_Act := FALSE;
	END_IF

	(* Unforce all Global *)
	IF (VIS2MM.tPlantComm.bFrc_Gbl) THEN
		(* Reset HMI Selection of Force Active *)
		FOR x:=0 TO tHmiDiag.iDiagTableSize-1 DO
			VIS2MM.tPlantComm.bFrc[x] := FALSE;
		END_FOR
		(* Unforce all Signals from/to all Masters*)
		FOR iAssetNum:=1 TO 4 DO
			(* Unforce Analog Inputs/Outputs *)
			FOR x:=0 TO tHmiDiag.iAnaSigCntE2M - 1 DO
				tPlantCom_M2E_In_Hmi[iAssetNum].bAnaForceActive[x] := FALSE;
				tPlantCom_E2M_Out_Hmi[iAssetNum].bAnaForceActive[x] := FALSE;
			END_FOR
			(* Unforce Digital Inputs/Outputs *)
			FOR x:=0 TO tHmiDiag.iDigSigCntE2M - 1 DO
				tPlantCom_M2E_In_Hmi[iAssetNum].bDigForceActive[x] := FALSE;
				tPlantCom_E2M_Out_Hmi[iAssetNum].bDigForceActive[x] := FALSE;
			END_FOR
			(* Set counter for forced signals to zero*)
			tPlantCom_M2E_In_Hmi[iAssetNum].iNum_ForcedValues 		:= 0;
			tPlantCom_E2M_Out_Hmi[iAssetNum].iNum_ForcedValues  	:= 0;
		END_FOR
		(* Unforce all Signals from/to all Engines *)
		FOR iAssetNum:=1 TO 32 DO
			(* Unforce Analog Inputs/Outputs *)
			FOR x:=0 TO tHmiDiag.iAnaSigCntE2E - 1 DO
				tPlantCom_E2E_In_Hmi[iAssetNum].bAnaForceActive[x] := FALSE;
				tPlantCom_E2E_Out_Hmi.bAnaForceActive[x] := FALSE;
			END_FOR
			(* Unforce Digital Inputs/Outputs *)
			FOR x:=0 TO tHmiDiag.iDigSigCntE2E - 1 DO
				tPlantCom_E2E_In_Hmi[iAssetNum].bDigForceActive[x] := FALSE;
				tPlantCom_E2E_Out_Hmi.bDigForceActive[x] := FALSE;
			END_FOR
			(* Set counter for forced signals to zero*)
			tPlantCom_E2E_In_Hmi[iAssetNum].iNum_ForcedValues 		:= 0;
			tPlantCom_E2E_Out_Hmi.iNum_ForcedValues  				:= 0;
		END_FOR
		VIS2MM.tPlantComm.bFrc_Gbl := FALSE;
	END_IF

	// evaluate number of datapoints depending on the selection to interate over the stored hmi values
	iNum_Datapoints := 0;

	(* Copy the selected Data to the internal diagnostic arrays to be displayed on the HMI *)
	CASE tHmiDiag.iIO_Typ_Dir OF
		NO_SELECTION: (* No Selection *)
		FROM_MASTER: (* Signals from Master *)
			IF (tHmiDiag.iIO_Typ_Dir_Num >= 1 AND tHmiDiag.iIO_Typ_Dir_Num <= 4) THEN
				CASE tHmiDiag.iIO_Typ OF

					NO_SELECTION: (* No Selection default *)

					PlantComm_AI: (* Analog Input *)

						(* Validate Start Index *)
						IF (VIS2MM.tPlantComm.iNum_Start > tHmiDiag.iAnaSigCntE2M - tHmiDiag.iDiagTableSize) THEN
							tHmiDiag.iStartIdx := tHmiDiag.iAnaSigCntE2M - tHmiDiag.iDiagTableSize;
							VIS2MM.tPlantComm.iNum_Start := tHmiDiag.iStartIdx;
						ELSE
							tHmiDiag.iStartIdx := VIS2MM.tPlantComm.iNum_Start;
						END_IF

						iNum_Datapoints := tHmiDiag.iAnaSigCntE2M;
						tHmiDiag.iCommentOffset := INT_TO_UINT(400);

						FOR x:=0 TO tHmiDiag.iDiagTableSize - 1 DO
							(* HMI Selection Change *)
							IF (tHmiDiag.bSelectionChange) THEN
								(* Force Active *)
								VIS2MM.tPlantComm.bFrc[x] := tPlantCom_M2E_In_Hmi[tHmiDiag.iIO_Typ_Dir_Num].bAnaForceActive[tHmiDiag.iStartIdx+x];
								(* Force Value *)
								VIS2MM.tPlantComm.rFrc_Int[x] := tPlantCom_M2E_In_Hmi[tHmiDiag.iIO_Typ_Dir_Num].rForceValue[tHmiDiag.iStartIdx+x];
								(* Signal Number *)
								MM2VIS.tPlantComm.iNum[x] := tHmiDiag.iStartIdx + x;
								(* Comment Nr *)
								MM2VIS.tPlantComm.iComment[x] := tHmiDiag.iCommentOffset + tHmiDiag.iStartIdx + x;
							END_IF
							(* No HMI Selection Change *)
							IF(NOT tHmiDiag.bSelectionChange) THEN
								(* Force changes from inactive to active *)
								IF (NOT tPlantCom_M2E_In_Hmi[tHmiDiag.iIO_Typ_Dir_Num].bAnaForceActive[tHmiDiag.iStartIdx+x] AND VIS2MM.tPlantComm.bFrc[x]) THEN
									tPlantCom_M2E_In_Hmi[tHmiDiag.iIO_Typ_Dir_Num].iNum_ForcedValues := tPlantCom_M2E_In_Hmi[tHmiDiag.iIO_Typ_Dir_Num].iNum_ForcedValues + 1;
									(* Force changes from active to inactive *)
								ELSIF (tPlantCom_M2E_In_Hmi[tHmiDiag.iIO_Typ_Dir_Num].bAnaForceActive[tHmiDiag.iStartIdx+x] AND NOT VIS2MM.tPlantComm.bFrc[x]) THEN
									tPlantCom_M2E_In_Hmi[tHmiDiag.iIO_Typ_Dir_Num].iNum_ForcedValues := tPlantCom_M2E_In_Hmi[tHmiDiag.iIO_Typ_Dir_Num].iNum_ForcedValues - 1;
								END_IF
								(* Store Force Variables *)
								tPlantCom_M2E_In_Hmi[tHmiDiag.iIO_Typ_Dir_Num].bAnaForceActive[tHmiDiag.iStartIdx+x] := VIS2MM.tPlantComm.bFrc[x];
								tPlantCom_M2E_In_Hmi[tHmiDiag.iIO_Typ_Dir_Num].rForceValue[tHmiDiag.iStartIdx+x] := VIS2MM.tPlantComm.rFrc_Int[x];
							END_IF

							(* Display Foced Value as Internal and Bus Value as External Signal when Signal is forced *)
							IF (VIS2MM.tPlantComm.bFrc[x]) THEN
								MM2VIS.tPlantComm.rInt[x] := tPlantCom_M2E_In_Hmi[tHmiDiag.iIO_Typ_Dir_Num].rForceValue[tHmiDiag.iStartIdx+x];
								MM2VIS.tPlantComm.rExt[x] := tPlantCom_M2E_In_Bus[tHmiDiag.iIO_Typ_Dir_Num].analogSignals[tHmiDiag.iStartIdx+x].Value;
							ELSE
							(* Display Bus Value as Externals and Internal Signal when Signal is not forced *)
								MM2VIS.tPlantComm.rExt[x] := tPlantCom_M2E_In_Bus[tHmiDiag.iIO_Typ_Dir_Num].analogSignals[tHmiDiag.iStartIdx+x].Value;
								MM2VIS.tPlantComm.rInt[x] := tPlantCom_M2E_In_Plc[tHmiDiag.iIO_Typ_Dir_Num].analogSignals[tHmiDiag.iStartIdx+x].Value;
							END_IF
						END_FOR

					PlantComm_DI: (* Digital Input *)
						(* Validate Start Index *)
						IF (VIS2MM.tPlantComm.iNum_Start > tHmiDiag.iDigSigCntE2M - tHmiDiag.iDiagTableSize) THEN
							tHmiDiag.iStartIdx := tHmiDiag.iDigSigCntE2M - tHmiDiag.iDiagTableSize;
							VIS2MM.tPlantComm.iNum_Start := tHmiDiag.iStartIdx;
						ELSE
							tHmiDiag.iStartIdx := VIS2MM.tPlantComm.iNum_Start;
						END_IF

						iNum_Datapoints := tHmiDiag.iDigSigCntE2M;
						tHmiDiag.iCommentOffset := INT_TO_UINT(100);

						FOR x:=0 TO tHmiDiag.iDiagTableSize - 1 DO
							(* Hmi Selection Change *)
							IF (tHmiDiag.bSelectionChange) THEN
								(* Force Active*)
								VIS2MM.tPlantComm.bFrc[x] := tPlantCom_M2E_In_Hmi[tHmiDiag.iIO_Typ_Dir_Num].bDigForceActive[tHmiDiag.iStartIdx+x];
								(* Force Value *)
								VIS2MM.tPlantComm.bFrc_Int[x] := tPlantCom_M2E_In_Hmi[tHmiDiag.iIO_Typ_Dir_Num].bForceValue[tHmiDiag.iStartIdx+x];
								(* Signal Number *)
								MM2VIS.tPlantComm.iNum[x] := tHmiDiag.iStartIdx + x;
								(* Comment Nr *)
								MM2VIS.tPlantComm.iComment[x] := tHmiDiag.iCommentOffset + tHmiDiag.iStartIdx + x;
							END_IF
							(* No HMI Selection change *)
							IF (NOT tHmiDiag.bSelectionChange) THEN
								(* Force changes from inactive to active *)
								IF (NOT tPlantCom_M2E_In_Hmi[tHmiDiag.iIO_Typ_Dir_Num].bDigForceActive[tHmiDiag.iStartIdx+x] AND VIS2MM.tPlantComm.bFrc[x]) THEN
									tPlantCom_M2E_In_Hmi[tHmiDiag.iIO_Typ_Dir_Num].iNum_ForcedValues := tPlantCom_M2E_In_Hmi[tHmiDiag.iIO_Typ_Dir_Num].iNum_ForcedValues + 1;
									(* Force changes from active to inactive *)
								ELSIF (tPlantCom_M2E_In_Hmi[tHmiDiag.iIO_Typ_Dir_Num].bDigForceActive[tHmiDiag.iStartIdx+x] AND NOT VIS2MM.tPlantComm.bFrc[x]) THEN
									tPlantCom_M2E_In_Hmi[tHmiDiag.iIO_Typ_Dir_Num].iNum_ForcedValues := tPlantCom_M2E_In_Hmi[tHmiDiag.iIO_Typ_Dir_Num].iNum_ForcedValues - 1;
								END_IF
								(* Store Force Values *)
								tPlantCom_M2E_In_Hmi[tHmiDiag.iIO_Typ_Dir_Num].bDigForceActive[tHmiDiag.iStartIdx+x] := VIS2MM.tPlantComm.bFrc[x];
								tPlantCom_M2E_In_Hmi[tHmiDiag.iIO_Typ_Dir_Num].bForceValue[tHmiDiag.iStartIdx+x] := VIS2MM.tPlantComm.bFrc_Int[x];
							END_IF

							(* Display Foced Value as Internal and Bus Value as External Signal when Signal is forced *)
							IF (VIS2MM.tPlantComm.bFrc[x]) THEN
								MM2VIS.tPlantComm.rInt[x] := BOOL_TO_REAL(tPlantCom_M2E_In_Hmi[tHmiDiag.iIO_Typ_Dir_Num].bForceValue[tHmiDiag.iStartIdx+x]);
								MM2VIS.tPlantComm.rExt[x] := BOOL_TO_REAL(tPlantCom_M2E_In_Bus[tHmiDiag.iIO_Typ_Dir_Num].digitalSignals[tHmiDiag.iStartIdx+x].Value);
							ELSE
								(* Display Bus Value as Externals and Internal Signal when Signal is not forced *)
								MM2VIS.tPlantComm.rExt[x] := BOOL_TO_REAL(tPlantCom_M2E_In_Bus[tHmiDiag.iIO_Typ_Dir_Num].digitalSignals[tHmiDiag.iStartIdx+x].Value);
								MM2VIS.tPlantComm.rInt[x] := BOOL_TO_REAL(tPlantCom_M2E_In_Plc[tHmiDiag.iIO_Typ_Dir_Num].digitalSignals[tHmiDiag.iStartIdx+x].Value);
							END_IF
						END_FOR

					PlantComm_AO: (* Analog Output n/a *)

					PlantComm_DO: (* Digital Output n/a *)
				END_CASE
			END_IF
		FROM_ENGINE: (* Signals from Engine *)
			IF (tHmiDiag.iIO_Typ_Dir_Num >= 1 AND tHmiDiag.iIO_Typ_Dir_Num <= 32) THEN
				CASE tHmiDiag.iIO_Typ OF
					NO_SELECTION: (* No Selection default *)

					PlantComm_AI: (* Analog Input *)
						(* Validate Start Index *)
						IF (VIS2MM.tPlantComm.iNum_Start > tHmiDiag.iAnaSigCntE2E - tHmiDiag.iDiagTableSize) THEN
							tHmiDiag.iStartIdx := tHmiDiag.iAnaSigCntE2E - tHmiDiag.iDiagTableSize;
							VIS2MM.tPlantComm.iNum_Start := tHmiDiag.iStartIdx;
						ELSE
							tHmiDiag.iStartIdx := VIS2MM.tPlantComm.iNum_Start;
						END_IF;

						tHmiDiag.iCommentOffset := INT_TO_UINT(500);
						iNum_Datapoints := tHmiDiag.iAnaSigCntE2E;

						FOR x:=0 TO tHmiDiag.iDiagTableSize - 1 DO
							(* HMI Selection Change *)
							IF (tHmiDiag.bSelectionChange) THEN
								(* Signal Number *)
								MM2VIS.tPlantComm.iNum[x] := tHmiDiag.iStartIdx + x;
								(* Force Active *)
								VIS2MM.tPlantComm.bFrc[x] := tPlantCom_E2E_In_Hmi[tHmiDiag.iIO_Typ_Dir_Num].bAnaForceActive[tHmiDiag.iStartIdx + x];
								(* Force Value *)
								VIS2MM.tPlantComm.rFrc_Int[x] := tPlantCom_E2E_In_Hmi[tHmiDiag.iIO_Typ_Dir_Num].rForceValue[tHmiDiag.iStartIdx + x];
								(* Comment Nr *)
								MM2VIS.tPlantComm.iComment[x] := tHmiDiag.iCommentOffset + tHmiDiag.iStartIdx + x;
							END_IF
							(* No HMI Selection Change *)
							IF (NOT tHmiDiag.bSelectionChange) THEN
								(* Force changes from inactive to active *)
								IF (NOT tPlantCom_E2E_In_Hmi[tHmiDiag.iIO_Typ_Dir_Num].bAnaForceActive[tHmiDiag.iStartIdx+x] AND VIS2MM.tPlantComm.bFrc[x]) THEN
									tPlantCom_E2E_In_Hmi[tHmiDiag.iIO_Typ_Dir_Num].iNum_ForcedValues := tPlantCom_E2E_In_Hmi[tHmiDiag.iIO_Typ_Dir_Num].iNum_ForcedValues + 1;
								(* Force changes from active to inactive *)
								ELSIF (tPlantCom_E2E_In_Hmi[tHmiDiag.iIO_Typ_Dir_Num].bAnaForceActive[tHmiDiag.iStartIdx+x] AND NOT VIS2MM.tPlantComm.bFrc[x]) THEN
									tPlantCom_E2E_In_Hmi[tHmiDiag.iIO_Typ_Dir_Num].iNum_ForcedValues := tPlantCom_E2E_In_Hmi[tHmiDiag.iIO_Typ_Dir_Num].iNum_ForcedValues - 1;
								END_IF

								(* Store Force Values *)
								tPlantCom_E2E_In_Hmi[tHmiDiag.iIO_Typ_Dir_Num].bAnaForceActive[tHmiDiag.iStartIdx+x] := VIS2MM.tPlantComm.bFrc[x];
								tPlantCom_E2E_In_Hmi[tHmiDiag.iIO_Typ_Dir_Num].rForceValue[tHmiDiag.iStartIdx+x] := VIS2MM.tPlantComm.rFrc_Int[x];
							END_IF

							(* Display Foced Value as Internal and Bus Value as External Signal when Signal is forced *)
							IF (VIS2MM.tPlantComm.bFrc[x]) THEN
								MM2VIS.tPlantComm.rInt[x] := tPlantCom_E2E_In_Hmi[tHmiDiag.iIO_Typ_Dir_Num].rForceValue[tHmiDiag.iStartIdx+x];
								MM2VIS.tPlantComm.rExt[x] := tPlantCom_E2E_In_Bus[tHmiDiag.iIO_Typ_Dir_Num].analogSignals[tHmiDiag.iStartIdx+x].Value;
							ELSE
								(* Display Bus Value as Externals and Internal Signal when Signal is not forced *)
								MM2VIS.tPlantComm.rExt[x] := tPlantCom_E2E_In_Bus[tHmiDiag.iIO_Typ_Dir_Num].analogSignals[tHmiDiag.iStartIdx+x].Value;
								MM2VIS.tPlantComm.rInt[x] := tPlantCom_E2E_In_Plc[tHmiDiag.iIO_Typ_Dir_Num].analogSignals[tHmiDiag.iStartIdx+x].Value;
							END_IF
						END_FOR

					PlantComm_DI: (* Digital Input *)
						(* Evaluate Start Index *)
						IF (VIS2MM.tPlantComm.iNum_Start > tHmiDiag.iDigSigCntE2E - tHmiDiag.iDiagTableSize) THEN
							tHmiDiag.iStartIdx := tHmiDiag.iDigSigCntE2E - tHmiDiag.iDiagTableSize;
							VIS2MM.tPlantComm.iNum_Start := tHmiDiag.iStartIdx;
						ELSE
							tHmiDiag.iStartIdx := VIS2MM.tPlantComm.iNum_Start;
						END_IF

						iNum_Datapoints := tHmiDiag.iDigSigCntE2E;
						tHmiDiag.iCommentOffset := INT_TO_UINT(200);

						FOR x:=0 TO tHmiDiag.iDiagTableSize - 1 DO
							(* HMI Selection Change *)
							IF (tHmiDiag.bSelectionChange) THEN
								(* Signal Number *)
								MM2VIS.tPlantComm.iNum[x] := tHmiDiag.iStartIdx + x;
								(* Force Active *)
								VIS2MM.tPlantComm.bFrc[x] := tPlantCom_E2E_In_Hmi[tHmiDiag.iIO_Typ_Dir_Num].bDigForceActive[tHmiDiag.iStartIdx + x];
								(* Force Value BOOL *)
								VIS2MM.tPlantComm.bFrc_Int[x] := tPlantCom_E2E_In_Hmi[tHmiDiag.iIO_Typ_Dir_Num].bForceValue[tHmiDiag.iStartIdx + x];
								(* Comment Nr *)
								MM2VIS.tPlantComm.iComment[x] := tHmiDiag.iCommentOffset + tHmiDiag.iStartIdx + x;
							END_IF
							(* No HMI Selection Change *)
							IF (NOT tHmiDiag.bSelectionChange) THEN
								(* Force changes from inactive to active *)
								IF (NOT tPlantCom_E2E_In_Hmi[tHmiDiag.iIO_Typ_Dir_Num].bDigForceActive[tHmiDiag.iStartIdx+x] AND VIS2MM.tPlantComm.bFrc[x]) THEN
									tPlantCom_E2E_In_Hmi[tHmiDiag.iIO_Typ_Dir_Num].iNum_ForcedValues := tPlantCom_E2E_In_Hmi[tHmiDiag.iIO_Typ_Dir_Num].iNum_ForcedValues + 1;
									(* Force changes from active to inactive *)
								ELSIF (tPlantCom_E2E_In_Hmi[tHmiDiag.iIO_Typ_Dir_Num].bDigForceActive[tHmiDiag.iStartIdx+x] AND NOT VIS2MM.tPlantComm.bFrc[x]) THEN
									tPlantCom_E2E_In_Hmi[tHmiDiag.iIO_Typ_Dir_Num].iNum_ForcedValues := tPlantCom_E2E_In_Hmi[tHmiDiag.iIO_Typ_Dir_Num].iNum_ForcedValues - 1;
								END_IF

								(* Store Force Values *)
								tPlantCom_E2E_In_Hmi[tHmiDiag.iIO_Typ_Dir_Num].bDigForceActive[tHmiDiag.iStartIdx+x] := VIS2MM.tPlantComm.bFrc[x];
								tPlantCom_E2E_In_Hmi[tHmiDiag.iIO_Typ_Dir_Num].bForceValue[tHmiDiag.iStartIdx+x] := VIS2MM.tPlantComm.bFrc_Int[x];
							END_IF

							(* Display Foced Value as Internal and Bus Value as External Signal when Signal is forced *)
							IF (VIS2MM.tPlantComm.bFrc[x]) THEN
								MM2VIS.tPlantComm.rInt[x] := BOOL_TO_REAL(tPlantCom_E2E_In_Hmi[tHmiDiag.iIO_Typ_Dir_Num].bForceValue[tHmiDiag.iStartIdx+x]);
								MM2VIS.tPlantComm.rExt[x] := BOOL_TO_REAL(tPlantCom_E2E_In_Bus[tHmiDiag.iIO_Typ_Dir_Num].digitalSignals[tHmiDiag.iStartIdx+x].Value);
							ELSE
								(* Display Bus Value as Externals and Internal Signal when Signal is not forced *)
								MM2VIS.tPlantComm.rExt[x] := BOOL_TO_REAL(tPlantCom_E2E_In_Bus[tHmiDiag.iIO_Typ_Dir_Num].digitalSignals[tHmiDiag.iStartIdx+x].Value);
								MM2VIS.tPlantComm.rInt[x] := BOOL_TO_REAL(tPlantCom_E2E_In_Plc[tHmiDiag.iIO_Typ_Dir_Num].digitalSignals[tHmiDiag.iStartIdx+x].Value);
							END_IF
						END_FOR

					PlantComm_AO: (* Analog Output n/a *)
					PlantComm_DO: (* Digital Output n/a *)
				END_CASE
			END_IF

		TO_MASTER: (* Signals to Master *)

			CASE tHmiDiag.iIO_Typ OF
				NO_SELECTION: (* No Selection default *)

				PlantComm_AI: (* Analog Input n/a *)

				PlantComm_DI: (* Digital Input n/a *)

				PlantComm_AO: (* Analog Output *)
					(* Validate Start Index *)
					IF (VIS2MM.tPlantComm.iNum_Start > tHmiDiag.iAnaSigCntE2M - tHmiDiag.iDiagTableSize) THEN
						tHmiDiag.iStartIdx := tHmiDiag.iAnaSigCntE2M - tHmiDiag.iDiagTableSize;
						VIS2MM.tPlantComm.iNum_Start := tHmiDiag.iStartIdx;
					ELSE
						tHmiDiag.iStartIdx := VIS2MM.tPlantComm.iNum_Start;
					END_IF;

					iNum_Datapoints := tHmiDiag.iAnaSigCntE2M;
					tHmiDiag.iCommentOffset := INT_TO_UINT(300);

					FOR x:=0 TO tHmiDiag.iDiagTableSize - 1 DO
						(* HMI Selection Change*)
						IF (tHmiDiag.bSelectionChange) THEN
							(* Force Active *)
							VIS2MM.tPlantComm.bFrc[x] := tPlantCom_E2M_Out_Hmi[tHmiDiag.iIO_Typ_Dir_Num].bAnaForceActive[tHmiDiag.iStartIdx+x];
							(* Force Value *)
							VIS2MM.tPlantComm.rFrc_Int[x] := tPlantCom_E2M_Out_Hmi[tHmiDiag.iIO_Typ_Dir_Num].rForceValue[tHmiDiag.iStartIdx+x];
							(* Signal Number *)
							MM2VIS.tPlantComm.iNum[x] := tHmiDiag.iStartIdx + x;
							(* Comment Nr *)
							MM2VIS.tPlantComm.iComment[x] := tHmiDiag.iCommentOffset + tHmiDiag.iStartIdx + x;
						END_IF
						(* No HMI Selection Change *)
						IF (NOT tHmiDiag.bSelectionChange) THEN
							(* Force changes from inactive to active *)
							IF (NOT tPlantCom_E2M_Out_Hmi[tHmiDiag.iIO_Typ_Dir_Num].bAnaForceActive[tHmiDiag.iStartIdx+x] AND VIS2MM.tPlantComm.bFrc[x]) THEN
								tPlantCom_E2M_Out_Hmi[tHmiDiag.iIO_Typ_Dir_Num].iNum_ForcedValues := tPlantCom_E2M_Out_Hmi[tHmiDiag.iIO_Typ_Dir_Num].iNum_ForcedValues + 1;
							(* Force changes from active to inactive *)
							ELSIF (tPlantCom_E2M_Out_Hmi[tHmiDiag.iIO_Typ_Dir_Num].bAnaForceActive[tHmiDiag.iStartIdx+x] AND NOT VIS2MM.tPlantComm.bFrc[x]) THEN
								tPlantCom_E2M_Out_Hmi[tHmiDiag.iIO_Typ_Dir_Num].iNum_ForcedValues := tPlantCom_E2M_Out_Hmi[tHmiDiag.iIO_Typ_Dir_Num].iNum_ForcedValues - 1;
							END_IF
							(* Store Force Value from HMI*)
							tPlantCom_E2M_Out_Hmi[tHmiDiag.iIO_Typ_Dir_Num].bAnaForceActive[tHmiDiag.iStartIdx+x] := VIS2MM.tPlantComm.bFrc[x];
							tPlantCom_E2M_Out_Hmi[tHmiDiag.iIO_Typ_Dir_Num].rForceValue[tHmiDiag.iStartIdx+x] := VIS2MM.tPlantComm.rFrc_Int[x];
						END_IF

						IF (VIS2MM.tPlantComm.bFrc[x]) THEN
							MM2VIS.tPlantComm.rExt[x] := tPlantCom_E2M_Out_Hmi[tHmiDiag.iIO_Typ_Dir_Num].rForceValue[tHmiDiag.iStartIdx+x];
							MM2VIS.tPlantComm.rInt[x] := tPlantCom_E2M_Out_Plc[tHmiDiag.iIO_Typ_Dir_Num].analogSignals[tHmiDiag.iStartIdx+x].Value;
						ELSE
							MM2VIS.tPlantComm.rExt[x] := tPlantCom_E2M_Out_Bus[tHmiDiag.iIO_Typ_Dir_Num].analogSignals[tHmiDiag.iStartIdx+x].Value;
							MM2VIS.tPlantComm.rInt[x] := tPlantCom_E2M_Out_Plc[tHmiDiag.iIO_Typ_Dir_Num].analogSignals[tHmiDiag.iStartIdx+x].Value;
						END_IF
					END_FOR

				PlantComm_DO: (* Digital Output *)
					(* Validate Start Index *)
					IF (VIS2MM.tPlantComm.iNum_Start > tHmiDiag.iDigSigCntE2M - tHmiDiag.iDiagTableSize) THEN
						tHmiDiag.iStartIdx := tHmiDiag.iDigSigCntE2M - tHmiDiag.iDiagTableSize;
						VIS2MM.tPlantComm.iNum_Start := tHmiDiag.iStartIdx;
					ELSE
						tHmiDiag.iStartIdx := VIS2MM.tPlantComm.iNum_Start;
					END_IF

					iNum_Datapoints := tHmiDiag.iDigSigCntE2M;
					tHmiDiag.iCommentOffset := INT_TO_UINT(0);

					FOR x:=0 TO tHmiDiag.iDiagTableSize - 1 DO
						(* HMI Selection Change *)
						IF (tHmiDiag.bSelectionChange) THEN
							(* Signal Number *)
							MM2VIS.tPlantComm.iNum[x] := tHmiDiag.iStartIdx + x;
							(* Force Active *)
							VIS2MM.tPlantComm.bFrc[x] := tPlantCom_E2M_Out_Hmi[tHmiDiag.iIO_Typ_Dir_Num].bDigForceActive[tHmiDiag.iStartIdx + x];
							(* Force Value BOOL *)
							VIS2MM.tPlantComm.bFrc_Int[x] := tPlantCom_E2M_Out_Hmi[tHmiDiag.iIO_Typ_Dir_Num].bForceValue[tHmiDiag.iStartIdx + x];
							(* Comment Nr *)
							MM2VIS.tPlantComm.iComment[x] := tHmiDiag.iCommentOffset + tHmiDiag.iStartIdx + x;
						END_IF
						(* No HMI Selection Change *)
						IF (NOT tHmiDiag.bSelectionChange) THEN
							(* Force changes from inactive to active *)
							IF (NOT tPlantCom_E2M_Out_Hmi[tHmiDiag.iIO_Typ_Dir_Num].bDigForceActive[tHmiDiag.iStartIdx+x] AND VIS2MM.tPlantComm.bFrc[x]) THEN
								tPlantCom_E2M_Out_Hmi[tHmiDiag.iIO_Typ_Dir_Num].iNum_ForcedValues := tPlantCom_E2M_Out_Hmi[tHmiDiag.iIO_Typ_Dir_Num].iNum_ForcedValues + 1;
								(* Force changes from active to inactive *)
							ELSIF (tPlantCom_E2M_Out_Hmi[tHmiDiag.iIO_Typ_Dir_Num].bDigForceActive[tHmiDiag.iStartIdx+x] AND NOT VIS2MM.tPlantComm.bFrc[x]) THEN
								tPlantCom_E2M_Out_Hmi[tHmiDiag.iIO_Typ_Dir_Num].iNum_ForcedValues := tPlantCom_E2M_Out_Hmi[tHmiDiag.iIO_Typ_Dir_Num].iNum_ForcedValues - 1;
							END_IF
							(* Store Force Values *)
							tPlantCom_E2M_Out_Hmi[tHmiDiag.iIO_Typ_Dir_Num].bDigForceActive[tHmiDiag.iStartIdx+x] := VIS2MM.tPlantComm.bFrc[x];
							tPlantCom_E2M_Out_Hmi[tHmiDiag.iIO_Typ_Dir_Num].bForceValue[tHmiDiag.iStartIdx+x] := VIS2MM.tPlantComm.bFrc_Int[x];
						END_IF

						IF (VIS2MM.tPlantComm.bFrc[x]) THEN
							MM2VIS.tPlantComm.rExt[x] := BOOL_TO_REAL(tPlantCom_E2M_Out_Hmi[tHmiDiag.iIO_Typ_Dir_Num].bForceValue[tHmiDiag.iStartIdx+x]);
							MM2VIS.tPlantComm.rInt[x] := BOOL_TO_REAL(tPlantCom_E2M_Out_Plc[tHmiDiag.iIO_Typ_Dir_Num].digitalSignals[tHmiDiag.iStartIdx+x].Value);
						ELSE
							MM2VIS.tPlantComm.rExt[x] := BOOL_TO_REAL(tPlantCom_E2M_Out_Bus[tHmiDiag.iIO_Typ_Dir_Num].digitalSignals[tHmiDiag.iStartIdx+x].Value);
							MM2VIS.tPlantComm.rInt[x] := BOOL_TO_REAL(tPlantCom_E2M_Out_Plc[tHmiDiag.iIO_Typ_Dir_Num].digitalSignals[tHmiDiag.iStartIdx+x].Value);
						END_IF
					END_FOR
			END_CASE
		TO_ENGINE: (* Signals to Engine*)
			CASE tHmiDiag.iIO_Typ OF
				NO_SELECTION: (* No Selection default *)

				PlantComm_AI: (* Analog Input n/a*)

				PlantComm_DI: (* Digital Input n/a*)

				PlantComm_AO: (* Analog Output *)
					(* Validate Start Index *)
					IF (VIS2MM.tPlantComm.iNum_Start > tHmiDiag.iAnaSigCntE2E - tHmiDiag.iDiagTableSize) THEN
						tHmiDiag.iStartIdx := tHmiDiag.iAnaSigCntE2E - tHmiDiag.iDiagTableSize;
						VIS2MM.tPlantComm.iNum_Start := tHmiDiag.iStartIdx;
					ELSE
						tHmiDiag.iStartIdx := VIS2MM.tPlantComm.iNum_Start;
					END_IF

					iNum_Datapoints := tHmiDiag.iAnaSigCntE2E;
					tHmiDiag.iCommentOffset := INT_TO_UINT(500);

					FOR x:=0 TO tHmiDiag.iDiagTableSize - 1 DO
						(* HMI Selection Change *)
						IF (tHmiDiag.bSelectionChange) THEN
							(* Force Active *)
							VIS2MM.tPlantComm.bFrc[x] := tPlantCom_E2E_Out_Hmi.bAnaForceActive[tHmiDiag.iStartIdx+x];
							(* Force Value *)
							VIS2MM.tPlantComm.rFrc_Int[x] := tPlantCom_E2E_Out_Hmi.rForceValue[tHmiDiag.iStartIdx+x];
							(* Signal Number *)
							MM2VIS.tPlantComm.iNum[x] := tHmiDiag.iStartIdx + x;
							(* Comment Nr *)
							MM2VIS.tPlantComm.iComment[x] := tHmiDiag.iCommentOffset + tHmiDiag.iStartIdx + x;
						END_IF
						(* No HMI Selection Change *)
						IF (NOT tHmiDiag.bSelectionChange) THEN
							(* Force changes from inactive to active *)
							IF (NOT tPlantCom_E2E_Out_Hmi.bAnaForceActive[tHmiDiag.iStartIdx+x] AND VIS2MM.tPlantComm.bFrc[x]) THEN
								tPlantCom_E2E_Out_Hmi.iNum_ForcedValues := tPlantCom_E2E_Out_Hmi.iNum_ForcedValues + 1;
							(* Force changes from active to inactive *)
							ELSIF (tPlantCom_E2E_Out_Hmi.bAnaForceActive[tHmiDiag.iStartIdx+x] AND NOT VIS2MM.tPlantComm.bFrc[x]) THEN
								tPlantCom_E2E_Out_Hmi.iNum_ForcedValues := tPlantCom_E2E_Out_Hmi.iNum_ForcedValues - 1;
							END_IF
							(* Store Forced Values *)
							tPlantCom_E2E_Out_Hmi.bAnaForceActive[tHmiDiag.iStartIdx+x] := VIS2MM.tPlantComm.bFrc[x];
							tPlantCom_E2E_Out_Hmi.rForceValue[tHmiDiag.iStartIdx+x] := VIS2MM.tPlantComm.rFrc_Int[x];
						END_IF

						IF (VIS2MM.tPlantComm.bFrc[x]) THEN
							MM2VIS.tPlantComm.rExt[x] := tPlantCom_E2E_Out_Hmi.rForceValue[tHmiDiag.iStartIdx+x];
							MM2VIS.tPlantComm.rInt[x] := tPlantCom_E2E_Out_Plc.analogSignals[tHmiDiag.iStartIdx+x].Value;
						ELSE
							MM2VIS.tPlantComm.rExt[x] := tPlantCom_E2E_Out_Bus.analogSignals[tHmiDiag.iStartIdx+x].Value;
							MM2VIS.tPlantComm.rInt[x] := tPlantCom_E2E_Out_Plc.analogSignals[tHmiDiag.iStartIdx+x].Value;
						END_IF
					END_FOR

				PlantComm_DO: (* Digital Output *)
					(* Evaluate Start Index *)
					IF (VIS2MM.tPlantComm.iNum_Start > tHmiDiag.iDigSigCntE2E - tHmiDiag.iDiagTableSize) THEN
						tHmiDiag.iStartIdx := tHmiDiag.iDigSigCntE2E - tHmiDiag.iDiagTableSize;
						VIS2MM.tPlantComm.iNum_Start := tHmiDiag.iStartIdx;
					ELSE
						tHmiDiag.iStartIdx := VIS2MM.tPlantComm.iNum_Start;
					END_IF

					iNum_Datapoints := tHmiDiag.iDigSigCntE2E;
					tHmiDiag.iCommentOffset := INT_TO_UINT(200);

					FOR x:=0 TO tHmiDiag.iDiagTableSize - 1 DO
						IF (tHmiDiag.bSelectionChange) THEN
							(* Force Active *)
							VIS2MM.tPlantComm.bFrc[x] := tPlantCom_E2E_Out_Hmi.bDigForceActive[tHmiDiag.iStartIdx+x];
							(* Force Value *)
							VIS2MM.tPlantComm.bFrc_Int[x] := tPlantCom_E2E_Out_Hmi.bForceValue[tHmiDiag.iStartIdx+x];
							(* Signal Number *)
							MM2VIS.tPlantComm.iNum[x] := tHmiDiag.iStartIdx + x;
							(* Comment Nr *)
							MM2VIS.tPlantComm.iComment[x] := tHmiDiag.iCommentOffset + tHmiDiag.iStartIdx + x;
						END_IF
						(* No HMI Selection Change *)
						IF (NOT tHmiDiag.bSelectionChange) THEN
							(* Force changes from inactive to active *)
							IF (NOT tPlantCom_E2E_Out_Hmi.bDigForceActive[tHmiDiag.iStartIdx+x] AND VIS2MM.tPlantComm.bFrc[x]) THEN
								tPlantCom_E2E_Out_Hmi.iNum_ForcedValues := tPlantCom_E2E_Out_Hmi.iNum_ForcedValues + 1;
							(* Force changes from active to inactive *)
							ELSIF (tPlantCom_E2E_Out_Hmi.bDigForceActive[tHmiDiag.iStartIdx+x] AND NOT VIS2MM.tPlantComm.bFrc[x]) THEN
								tPlantCom_E2E_Out_Hmi.iNum_ForcedValues := tPlantCom_E2E_Out_Hmi.iNum_ForcedValues - 1;
							END_IF
							(* Store Force Value *)
							tPlantCom_E2E_Out_Hmi.bDigForceActive[tHmiDiag.iStartIdx+x] := VIS2MM.tPlantComm.bFrc[x];
							tPlantCom_E2E_Out_Hmi.bForceValue[tHmiDiag.iStartIdx+x] := VIS2MM.tPlantComm.bFrc_Int[x];
						END_IF

						IF (VIS2MM.tPlantComm.bFrc[x]) THEN
							MM2VIS.tPlantComm.rExt[x] := BOOL_TO_REAL(tPlantCom_E2E_Out_Hmi.bForceValue[tHmiDiag.iStartIdx+x]);
							MM2VIS.tPlantComm.rInt[x] := BOOL_TO_REAL(tPlantCom_E2E_Out_Plc.digitalSignals[tHmiDiag.iStartIdx+x].Value);
						ELSE
							MM2VIS.tPlantComm.rExt[x] := BOOL_TO_REAL(tPlantCom_E2E_Out_Bus.digitalSignals[tHmiDiag.iStartIdx+x].Value);
							MM2VIS.tPlantComm.rInt[x] := BOOL_TO_REAL(tPlantCom_E2E_Out_Plc.digitalSignals[tHmiDiag.iStartIdx+x].Value);
						END_IF
					END_FOR
			END_CASE
	END_CASE

	(* Calculate the number of forced values for the selected Asset *)
	MM2VIS.tPlantComm.iFrc_Act := 0;
	(* Check if an Asset is selected *)
	IF (tHmiDiag.iIO_Typ_Dir_Num >= 1 AND tHmiDiag.iIO_Typ_Dir_Num <= 4) THEN
		IF (tHmiDiag.iIO_Typ_Dir = FROM_MASTER OR tHmiDiag.iIO_Typ_Dir = TO_MASTER) THEN
			(* Number of Forced Analog Inputs/Outputs *)
			FOR x:=0 TO tHmiDiag.iAnaSigCntE2M - 1 DO
				IF (tPlantCom_M2E_In_Hmi[tHmiDiag.iIO_Typ_Dir_Num].bAnaForceActive[x]) THEN
					MM2VIS.tPlantComm.iFrc_Act := MM2VIS.tPlantComm.iFrc_Act + 1;
				END_IF
				IF (tPlantCom_E2M_Out_Hmi[tHmiDiag.iIO_Typ_Dir_Num].bAnaForceActive[x]) THEN
					MM2VIS.tPlantComm.iFrc_Act := MM2VIS.tPlantComm.iFrc_Act + 1;
				END_IF
			END_FOR
			(* Number of Forced Digital Inputs/Outputs *)
			FOR x:=0 TO tHmiDiag.iDigSigCntE2M - 1 DO
				IF (tPlantCom_M2E_In_Hmi[tHmiDiag.iIO_Typ_Dir_Num].bDigForceActive[x]) THEN
					MM2VIS.tPlantComm.iFrc_Act := MM2VIS.tPlantComm.iFrc_Act + 1;
				END_IF

				IF (tPlantCom_E2M_Out_Hmi[tHmiDiag.iIO_Typ_Dir_Num].bDigForceActive[x]) THEN
					MM2VIS.tPlantComm.iFrc_Act := MM2VIS.tPlantComm.iFrc_Act + 1;
				END_IF
			END_FOR
		ELSIF (tHmiDiag.iIO_Typ_Dir = FROM_ENGINE OR tHmiDiag.iIO_Typ_Dir = TO_ENGINE) THEN
			(* Number of Forced Analog Inputs/Outputs *)
			FOR x:=0 TO tHmiDiag.iAnaSigCntE2E - 1 DO
				IF (tPlantCom_E2E_In_Hmi[tHmiDiag.iIO_Typ_Dir_Num].bAnaForceActive[x]) THEN
					MM2VIS.tPlantComm.iFrc_Act := MM2VIS.tPlantComm.iFrc_Act + 1;
				END_IF
				IF (tPlantCom_E2E_Out_Hmi.bAnaForceActive[x]) THEN
					MM2VIS.tPlantComm.iFrc_Act := MM2VIS.tPlantComm.iFrc_Act + 1;
				END_IF
			END_FOR
			(* Number of Forced Digital Inputs/Outputs *)
			FOR x:=0 TO tHmiDiag.iDigSigCntE2E - 1 DO
				IF (tPlantCom_E2E_In_Hmi[tHmiDiag.iIO_Typ_Dir_Num].bDigForceActive[x]) THEN
					MM2VIS.tPlantComm.iFrc_Act := MM2VIS.tPlantComm.iFrc_Act + 1;
				END_IF
				IF (tPlantCom_E2E_Out_Hmi.bDigForceActive[x]) THEN
					MM2VIS.tPlantComm.iFrc_Act := MM2VIS.tPlantComm.iFrc_Act + 1;
				END_IF
			END_FOR
		END_IF
	END_IF

	(* Calculate the number of global forced values *)
	tHmiDiag.iForcedValueCntGlobal := 0;
	FOR x:=iMasNumMin TO iMasNumMax DO
		IF (x >= 1 AND x <= 4) THEN
			tHmiDiag.iForcedValueCntGlobal := tHmiDiag.iForcedValueCntGlobal + tPlantCom_M2E_In_Hmi[x].iNum_ForcedValues;
			tHmiDiag.iForcedValueCntGlobal := tHmiDiag.iForcedValueCntGlobal + tPlantCom_E2M_Out_Hmi[x].iNum_ForcedValues;
		END_IF
	END_FOR;

	FOR x:=iEngNumMin TO iEngNumMax DO
		IF (x >= 1 AND x <= 32) THEN
			tHmiDiag.iForcedValueCntGlobal := tHmiDiag.iForcedValueCntGlobal + tPlantCom_E2E_In_Hmi[x].iNum_ForcedValues;
		END_IF
	END_FOR;
	tHmiDiag.iForcedValueCntGlobal := tHmiDiag.iForcedValueCntGlobal + tPlantCom_E2E_Out_Hmi.iNum_ForcedValues;
	MM2VIS.tPlantComm.iFrc_Gbl := tHmiDiag.iForcedValueCntGlobal;

	(* Initial Value of the comment column on the hmi when nothing is selected *)
	IF (VIS2MM.tPlantComm.iIO_Typ = 0 OR VIS2MM.tPlantComm.iIO_Typ_Dir = 0) THEN
		FOR x:=0 TO tHmiDiag.iDiagTableSize-1 DO
			MM2VIS.tPlantComm.iFrc_Act := 0;
			MM2VIS.tPlantComm.iNum[x] := 0;
			MM2VIS.tPlantComm.rInt[x] := 0.0;
			MM2VIS.tPlantComm.rExt[x] := 0.0;
			MM2VIS.tPlantComm.iComment[x] := 99;
			VIS2MM.tPlantComm.bFrc[x] := FALSE;
			VIS2MM.tPlantComm.bFrc_Int[x] := FALSE;
			VIS2MM.tPlantComm.rFrc_Int[x] := 0.0;
		END_FOR
	END_IF

END_PROGRAM
```

#### Init.st - Init code
```iecst
(*******************************************************************************
Hmi Logic for the Plant Communication Diagnostics and Forcing screen

This code is confidential and proprietary to the INNIO Company.
It may not be used in any form, or reproduced in any manner, without the express
written permission of the INNIO Company.
Copyright, INNIO Company, 2024

Customized modifications: -
------------------------

History:
-------
V4.14.0	26.11.2024	Astner	Created Task

Instructions for use: -
--------------------

Outstandings:
------------

*******************************************************************************)

PROGRAM _INIT

	tHmiDiag.iAnaSigCntE2E := iAnaArrayMaxAll + 1;
	tHmiDiag.iDigSigCntE2E := iDigArrayMaxAll + 1;
	tHmiDiag.iAnaSigCntE2M := iAnaArrayMaxAll + 1;
	tHmiDiag.iDigSigCntE2M := iDigArrayMaxAll + 1;
	tHmiDiag.iDiagTableSize := 16;

END_PROGRAM
```

#### Types.typ - Local data types
```iecst
TYPE
	tHmiDiagnosticVariables : 	STRUCT  (*Holds variables needed for the HMI Force Screen Logic*)
		rInternalSignals : ARRAY[0..15]OF REAL;
		rExternalSignals : ARRAY[0..15]OF REAL;
		iIO_Typ : USINT;
		iIO_Typ_Dir : USINT;
		iIO_Typ_Dir_Num : USINT;
		iStartIdx : USINT;
		bForceActive : ARRAY[0..15]OF REAL;
		iDisplayNr : ARRAY[0..15]OF USINT;
		rForceValue : ARRAY[0..15]OF REAL;
		iCommentNr : UINT;
		iForcedValueCntGlobal : USINT;
		iAnaSigCntE2E : USINT;
		iDiagTableSize : USINT;
		iAnaSigCntE2M : USINT;
		iDigSigCntE2M : USINT;
		iDigSigCntE2E : USINT;
		iCommentOffset : UINT;
		bSelectionChange : BOOL;
		iForcedValueCntAsset_HMI : USINT;
	END_STRUCT;
END_TYPE
```

#### Variables.var - Local variables
```iecst
(*Selection Constants*)
VAR CONSTANT
	NO_SELECTION : USINT := 0;
	FROM_MASTER : USINT := 1;
	TO_MASTER : USINT := 3;
	FROM_ENGINE : USINT := 2;
	TO_ENGINE : USINT := 4;
	PlantComm_DI : USINT := 2;
	PlantComm_AI : USINT := 1;
	PlantComm_DO : USINT := 4;
	PlantComm_AO : USINT := 3;
END_VAR
(*Variables for the HMI Logic*)
VAR
	tHmiDiag : tHmiDiagnosticVariables := (0);
	x : USINT := 0;
	iNum_Datapoints : USINT := 0;
	iAssetNum : USINT := 0;
END_VAR
```

### Program Logical/HalIO/PlantCommunication/xComMapIn10ms (IEC, version 4.14.0)

#### InCyclic.st - Cyclic code
```iecst
(*******************************************************************************
Mapping from Bus Arrays to Plc Arrays with force logic

This code is confidential and proprietary to the INNIO Company.
It may not be used in any form, or reproduced in any manner, without the express
written permission of the INNIO Company.
Copyright, INNIO Company, 2024

Customized modifications: -
------------------------

History:
-------
V4.14.0	26.11.2024	Astner	Created Task

Instructions for use: -
--------------------

Outstandings:
------------

*******************************************************************************)
PROGRAM _CYCLIC
	(* Exit if configuration fails or not active *)

	IF (NOT MM2VIS.tPlantComm.bCfg_OK OR NOT Para.tPlantComm.bActive) THEN
		RETURN;
	END_IF

	(*************************************)
	(* Merge data from fast input arrays *)
	(*************************************)

	(*** Input from Engines  ***)
	FOR x:=iEngNumMin TO iEngNumMax DO
		memcpy(ADR(tPlantCom_E2E_In_Bus[x].digitalSignals[iDigArrayMax100ms+1]), ADR(tPlantCom_E2E_In_10ms[x].digitalSignals[0]), (iDigArrayMax10ms+1) * SIZEOF(tPlantCom_E2E_In_10ms[x].digitalSignals[0]));
		memcpy(ADR(tPlantCom_E2E_In_Bus[x].analogSignals[iAnaArrayMax100ms+1]), ADR(tPlantCom_E2E_In_10ms[x].analogSignals[0]), (iAnaArrayMax10ms+1) * SIZEOF(tPlantCom_E2E_In_10ms[x].analogSignals[0]));
	END_FOR;

	(*** Input from Masters  ***)
	FOR x:=iMasNumMin TO iMasNumMax DO
		memcpy(ADR(tPlantCom_M2E_In_Bus[x].digitalSignals[iDigArrayMax100ms+1]), ADR(tPlantCom_M2E_In_10ms[x].digitalSignals[0]), (iDigArrayMax10ms+1) * SIZEOF(tPlantCom_M2E_In_10ms[x].digitalSignals[0]));
		memcpy(ADR(tPlantCom_M2E_In_Bus[x].analogSignals[iAnaArrayMax100ms+1]), ADR(tPlantCom_M2E_In_10ms[x].analogSignals[0]), (iAnaArrayMax10ms+1) * SIZEOF(tPlantCom_M2E_In_10ms[x].analogSignals[0]));
	END_FOR;

	(***************************)
	(* Copy Data to Plc Arrays *)
	(***************************)

	(*** Fast Inputs from Engines  ***)
	FOR x:=iEngNumMin TO iEngNumMax DO
		memcpy(ADR(tPlantCom_E2E_In_Plc[x].digitalSignals[iDigArrayMax100ms+1]), ADR(tPlantCom_E2E_In_Bus[x].digitalSignals[iDigArrayMax100ms+1]), (iDigArrayMax10ms+1) * SIZEOF(tPlantCom_E2E_In_Plc[x].digitalSignals[0]));
		memcpy(ADR(tPlantCom_E2E_In_Plc[x].analogSignals[iAnaArrayMax100ms+1]), ADR(tPlantCom_E2E_In_Bus[x].analogSignals[iAnaArrayMax100ms+1]), (iAnaArrayMax10ms+1) * SIZEOF(tPlantCom_E2E_In_Plc[x].analogSignals[0]));
	END_FOR

	(*** Fast Inputs from Masters  ***)
	FOR x:=iMasNumMin TO iMasNumMax DO
		memcpy(ADR(tPlantCom_M2E_In_Plc[x].digitalSignals[iDigArrayMax100ms+1]), ADR(tPlantCom_M2E_In_Bus[x].digitalSignals[iDigArrayMax100ms+1]), (iDigArrayMax10ms+1) * SIZEOF(tPlantCom_M2E_In_Bus[x].digitalSignals[0]));
		memcpy(ADR(tPlantCom_M2E_In_Plc[x].analogSignals[iAnaArrayMax100ms+1]), ADR(tPlantCom_M2E_In_Bus[x].analogSignals[iAnaArrayMax100ms+1]), (iAnaArrayMax10ms+1) * SIZEOF(tPlantCom_M2E_In_Bus[x].analogSignals[0]));
	END_FOR;

	(* Skip overwriting with forced values if no signal is forced *)
	IF (MM2VIS.tPlantComm.iFrc_Gbl = 0) THEN
		RETURN;
	END_IF

	(***********************************************)
	(* Overwrite forced inputs with value from HMI *)
	(***********************************************)
	FOR x:=iEngNumMin TO iEngNumMax DO
		IF (tPlantCom_E2E_In_Hmi[x].iNum_ForcedValues > 0) THEN
			(* Fast Digital Signals *)
			FOR idx:=iDigArrayMax100ms+1 TO iDigArrayMaxAll DO
				IF (tPlantCom_E2E_In_Hmi[x].bDigForceActive[idx]) THEN
					tPlantCom_E2E_In_Plc[x].digitalSignals[idx].Value := tPlantCom_E2E_In_Hmi[x].bForceValue[idx];
					tPlantCom_E2E_In_Plc[x].digitalSignals[idx].GoodQual := TRUE;
				END_IF
			END_FOR
			(* Fast Analog Signals *)
			FOR idx:=iAnaArrayMax100ms+1 TO iAnaArrayMaxAll DO
				IF (tPlantCom_E2E_In_Hmi[x].bAnaForceActive[idx]) THEN
					tPlantCom_E2E_In_Plc[x].analogSignals[idx].Value := tPlantCom_E2E_In_Hmi[x].rForceValue[idx];
					tPlantCom_E2E_In_Plc[x].analogSignals[idx].GoodQual := TRUE;
				END_IF
			END_FOR
		END_IF
	END_FOR

	FOR x:=iMasNumMin TO iMasNumMax DO
		IF (tPlantCom_M2E_In_Hmi[x].iNum_ForcedValues > 0) THEN
			(* Fast Digital Signals *)
			FOR idx:=iDigArrayMax100ms+1 TO iDigArrayMaxAll DO
				IF (tPlantCom_M2E_In_Hmi[x].bDigForceActive[idx]) THEN
					tPlantCom_M2E_In_Plc[x].digitalSignals[idx].Value := tPlantCom_M2E_In_Hmi[x].bForceValue[idx];
					tPlantCom_M2E_In_Plc[x].digitalSignals[idx].GoodQual := TRUE;
				END_IF
			END_FOR
			(* Fast Analog Signals *)
			FOR idx:=iAnaArrayMax100ms+1 TO iAnaArrayMaxAll DO
				IF (tPlantCom_M2E_In_Hmi[x].bAnaForceActive[idx]) THEN
					tPlantCom_M2E_In_Plc[x].analogSignals[idx].Value := tPlantCom_M2E_In_Hmi[x].rForceValue[idx];
					tPlantCom_M2E_In_Plc[x].analogSignals[idx].GoodQual := TRUE;
				END_IF
			END_FOR
		END_IF
	END_FOR
END_PROGRAM
```

#### InInit.st - Init code
```iecst
(*******************************************************************************
Mapping from Bus Arrays to Plc Arrays with force logic

This code is confidential and proprietary to the INNIO Company.
It may not be used in any form, or reproduced in any manner, without the express
written permission of the INNIO Company.
Copyright, INNIO Company, 2024

Customized modifications: -
------------------------

History:
-------
V4.14.0	26.11.2024	Astner	Created Task

Instructions for use: -
--------------------

Outstandings:
------------

*******************************************************************************)

PROGRAM _INIT
	(* Insert code here *)

END_PROGRAM
```

#### InVariables.var - Local variables
```iecst
VAR
	idx : USINT := 0;
	x : USINT := 0;
END_VAR
```

### Program Logical/HalIO/PlantCommunication/xComMapIn100ms (IEC, version 4.14.0)

#### InCyclic.st - Cyclic code
```iecst
(*******************************************************************************
Mapping from Bus Arrays to Plc Arrays with force logic

This code is confidential and proprietary to the INNIO Company.
It may not be used in any form, or reproduced in any manner, without the express
written permission of the INNIO Company.
Copyright, INNIO Company, 2024

Customized modifications: -
------------------------

History:
-------
V4.14.0	26.11.2024	Astner	Created Task

Instructions for use: -
--------------------

Outstandings:
------------

*******************************************************************************)
PROGRAM _CYCLIC
	(* Exit if configuration fails or not active *)
	IF (NOT MM2VIS.tPlantComm.bCfg_OK OR NOT Para.tPlantComm.bActive) THEN
		RETURN;
	END_IF;
	(****************************************)
	(* Merge data from slow bus input array *)
	(****************************************)

	(*** Input from Engines  ***)
	FOR x:=iEngNumMin TO iEngNumMax DO
		memcpy(ADR(tPlantCom_E2E_In_Bus[x].digitalSignals[0]), ADR(tPlantCom_E2E_In_100ms[x].digitalSignals[0]), (iDigArrayMax100ms+1) * SIZEOF(tPlantCom_E2E_In_100ms[x].digitalSignals[0]));
		memcpy(ADR(tPlantCom_E2E_In_Bus[x].analogSignals[0]), ADR(tPlantCom_E2E_In_100ms[x].analogSignals[0]), (iAnaArrayMax100ms+1) * SIZEOF(tPlantCom_E2E_In_100ms[x].analogSignals[0]));
	END_FOR

	(*** Input from Masters  ***)
	FOR x:=iMasNumMin TO iMasNumMax DO
		memcpy(ADR(tPlantCom_M2E_In_Bus[x].digitalSignals[0]), ADR(tPlantCom_M2E_In_100ms[x].digitalSignals[0]), (iDigArrayMax100ms+1) * SIZEOF(tPlantCom_M2E_In_100ms[x].digitalSignals[0]));
		memcpy(ADR(tPlantCom_M2E_In_Bus[x].analogSignals[0]), ADR(tPlantCom_M2E_In_100ms[x].analogSignals[0]), (iAnaArrayMax100ms+1) * SIZEOF(tPlantCom_M2E_In_100ms[x].analogSignals[0]));
	END_FOR

	(***************************)
	(* Copy Data to Plc Arrays *)
	(***************************)

	(*** Input from Engines  ***)
	FOR x:=iEngNumMin TO iEngNumMax DO
		memcpy(ADR(tPlantCom_E2E_In_Plc[x].digitalSignals[0]), ADR(tPlantCom_E2E_In_Bus[x].digitalSignals[0]), (iDigArrayMax100ms+1) * SIZEOF(tPlantCom_E2E_In_Plc[x].digitalSignals[0]));
		memcpy(ADR(tPlantCom_E2E_In_Plc[x].analogSignals[0]), ADR(tPlantCom_E2E_In_Bus[x].analogSignals[0]), (iAnaArrayMax100ms+1) * SIZEOF(tPlantCom_E2E_In_Plc[x].analogSignals[0]));
	END_FOR

	(*** Input from Masters  ***)
	FOR x:=iMasNumMin TO iMasNumMax DO
		memcpy(ADR(tPlantCom_M2E_In_Plc[x].digitalSignals[0]), ADR(tPlantCom_M2E_In_Bus[x].digitalSignals[0]), (iDigArrayMax100ms+1) * SIZEOF(tPlantCom_M2E_In_Plc[x].digitalSignals[0]));
		memcpy(ADR(tPlantCom_M2E_In_Plc[x].analogSignals[0]), ADR(tPlantCom_M2E_In_Bus[x].analogSignals[0]), (iAnaArrayMax100ms+1) * SIZEOF(tPlantCom_M2E_In_Plc[x].analogSignals[0]));
	END_FOR;

	(* Skip overwriting with forced values if no signal is forced *)
	IF (MM2VIS.tPlantComm.iFrc_Gbl = 0) THEN
		RETURN;
	END_IF

	(***********************************************)
	(* Overwrite forced inputs with value from HMI *)
	(***********************************************)
	FOR x:=iEngNumMin TO iEngNumMax DO
		IF (tPlantCom_E2E_In_Hmi[x].iNum_ForcedValues > 0) THEN
			(* Digital Signals *)
			FOR idx:=0 TO iDigArrayMax100ms DO
				IF (tPlantCom_E2E_In_Hmi[x].bDigForceActive[idx]) THEN
					tPlantCom_E2E_In_Plc[x].digitalSignals[idx].Value := tPlantCom_E2E_In_Hmi[x].bForceValue[idx];
					tPlantCom_E2E_In_Plc[x].digitalSignals[idx].GoodQual := TRUE;
				END_IF
			END_FOR
			(* Analog Signals *)
			FOR idx:=0 TO iAnaArrayMax100ms DO
				IF (tPlantCom_E2E_In_Hmi[x].bAnaForceActive[idx]) THEN
					tPlantCom_E2E_In_Plc[x].analogSignals[idx].Value := tPlantCom_E2E_In_Hmi[x].rForceValue[idx];
					tPlantCom_E2E_In_Plc[x].analogSignals[idx].GoodQual := TRUE;
				END_IF
			END_FOR
		END_IF
	END_FOR

	FOR x:=iMasNumMin TO iMasNumMax DO
		IF (tPlantCom_M2E_In_Hmi[x].iNum_ForcedValues > 0) THEN
			(* Digital Signals *)
			FOR idx:=0 TO iDigArrayMax100ms DO
				IF (tPlantCom_M2E_In_Hmi[x].bDigForceActive[idx]) THEN
					tPlantCom_M2E_In_Plc[x].digitalSignals[idx].Value := tPlantCom_M2E_In_Hmi[x].bForceValue[idx];
					tPlantCom_M2E_In_Plc[x].digitalSignals[idx].GoodQual := TRUE;
				END_IF
			END_FOR
			(* Analog Signals *)
			FOR idx:=0 TO iAnaArrayMax100ms DO
				IF (tPlantCom_M2E_In_Hmi[x].bAnaForceActive[idx]) THEN
					tPlantCom_M2E_In_Plc[x].analogSignals[idx].Value := tPlantCom_M2E_In_Hmi[x].rForceValue[idx];
					tPlantCom_M2E_In_Plc[x].analogSignals[idx].GoodQual := TRUE;
				END_IF
			END_FOR
		END_IF
	END_FOR
END_PROGRAM
```

#### InInit.st - Init code
```iecst
(*******************************************************************************
Mapping from Bus Arrays to Plc Arrays with force logic

This code is confidential and proprietary to the INNIO Company.
It may not be used in any form, or reproduced in any manner, without the express
written permission of the INNIO Company.
Copyright, INNIO Company, 2024

Customized modifications: -
------------------------

History:
-------
V4.14.0	26.11.2024	Astner	Created Task

Instructions for use: -
--------------------

Outstandings:
------------

*******************************************************************************)

PROGRAM _INIT
	(* Insert code here *)

END_PROGRAM
```

#### InVariables.var - Local variables
```iecst
VAR
	idx : USINT := 0;
	x : USINT := 0;
END_VAR
```

### Program Logical/HalIO/PlantCommunication/xComMapOut10ms (IEC, version 4.14.0)

#### OutCyclic.st - Cyclic code
```iecst
(*******************************************************************************
Mapping from Plc Arrays to Bus Arrays with force logic

This code is confidential and proprietary to the INNIO Company.
It may not be used in any form, or reproduced in any manner, without the express
written permission of the INNIO Company.
Copyright, INNIO Company, 2024

Customized modifications: -
------------------------

History:
-------
V4.14.0	26.11.2024	Astner	Created Task

Instructions for use: -
--------------------

Outstandings:
------------

*******************************************************************************)
PROGRAM _CYCLIC
	(* Exit if configuration fails or not active *)
	IF (NOT MM2VIS.tPlantComm.bCfg_OK OR NOT Para.tPlantComm.bActive) THEN
		RETURN;
	END_IF;

	(***************************)
	(* Copy Data to Bus Arrays *)
	(***************************)

	(*** Output to Engines  ***)
	memcpy(ADR(tPlantCom_E2E_Out_Bus.digitalSignals[iDigArrayMax100ms+1]), ADR(tPlantCom_E2E_Out_Plc.digitalSignals[iDigArrayMax100ms+1]), (iDigArrayMax10ms+1) * SIZEOF(tPlantCom_E2E_Out_Bus.digitalSignals[0]));
	memcpy(ADR(tPlantCom_E2E_Out_Bus.analogSignals[iAnaArrayMax100ms+1]), ADR(tPlantCom_E2E_Out_Plc.analogSignals[iAnaArrayMax100ms+1]), (iAnaArrayMax10ms+1) * SIZEOF(tPlantCom_E2E_Out_Bus.analogSignals[0]));

	(*** Outputs to Masters  ***)
	FOR x:=iMasNumMin TO iMasNumMax DO
		memcpy(ADR(tPlantCom_E2M_Out_Bus[x].digitalSignals[iDigArrayMax100ms+1]), ADR(tPlantCom_E2M_Out_Plc[x].digitalSignals[iDigArrayMax100ms+1]), (iDigArrayMax10ms+1) * SIZEOF(tPlantCom_E2M_Out_Bus[x].digitalSignals[0]));
		memcpy(ADR(tPlantCom_E2M_Out_Bus[x].analogSignals[iAnaArrayMax100ms+1]), ADR(tPlantCom_E2M_Out_Plc[x].analogSignals[iAnaArrayMax100ms+1]), (iAnaArrayMax10ms+1) * SIZEOF(tPlantCom_E2M_Out_Bus[x].analogSignals[0]));
	END_FOR

	(************************************************)
	(* Overwrite forced outputs with value from HMI *)
	(************************************************)

	IF (MM2VIS.tPlantComm.iFrc_Gbl > 0) THEN
		IF (tPlantCom_E2E_Out_Hmi.iNum_ForcedValues > 0) THEN
			(* Digital Signals *)
			FOR idx:=iDigArrayMax100ms+1 TO iDigArrayMaxAll DO
				IF (tPlantCom_E2E_Out_Hmi.bDigForceActive[idx]) THEN
					tPlantCom_E2E_Out_Bus.digitalSignals[idx].Value := tPlantCom_E2E_Out_Hmi.bForceValue[idx];
					tPlantCom_E2E_Out_Bus.digitalSignals[idx].GoodQual := TRUE;
				END_IF
			END_FOR
			(* Analog Signals *)
			FOR idx:=iAnaArrayMax100ms+1 TO iAnaArrayMaxAll DO
				IF (tPlantCom_E2E_Out_Hmi.bAnaForceActive[idx]) THEN
					tPlantCom_E2E_Out_Bus.analogSignals[idx].Value := tPlantCom_E2E_Out_Hmi.rForceValue[idx];
					tPlantCom_E2E_Out_Bus.analogSignals[idx].GoodQual := TRUE;
				END_IF
			END_FOR
		END_IF

		FOR x:=iMasNumMin TO iMasNumMax DO
			IF (tPlantCom_E2M_Out_Hmi[x].iNum_ForcedValues > 0) THEN
				(* Digital Signals *)
				FOR idx:=iDigArrayMax100ms+1 TO iDigArrayMaxAll DO
					IF (tPlantCom_E2M_Out_Hmi[x].bDigForceActive[idx]) THEN
						tPlantCom_E2M_Out_Bus[x].digitalSignals[idx].Value := tPlantCom_E2M_Out_Hmi[x].bForceValue[idx];
						tPlantCom_E2M_Out_Bus[x].digitalSignals[idx].GoodQual := TRUE;
					END_IF
				END_FOR
				(* Analog Signals *)
				FOR idx:=iAnaArrayMax100ms TO iAnaArrayMaxAll DO
					IF (tPlantCom_E2M_Out_Hmi[x].bAnaForceActive[idx]) THEN
						tPlantCom_E2M_Out_Bus[x].analogSignals[idx].Value := tPlantCom_E2M_Out_Hmi[x].rForceValue[idx];
						tPlantCom_E2M_Out_Bus[x].analogSignals[idx].GoodQual := TRUE;
					END_IF
				END_FOR
			END_IF
		END_FOR
	END_IF

	(***************************************)
	(* Split data to 10ms and 100ms arrays *)
	(***************************************)

	(*** Output to Engines  ***)
	memcpy(ADR(tPlantCom_E2E_Out_10ms.digitalSignals), ADR(tPlantCom_E2E_Out_Bus.digitalSignals[iDigArrayMax100ms+1]), (iDigArrayMax10ms+1) * SIZEOF(tPlantCom_E2E_Out_10ms.digitalSignals[0]));
	memcpy(ADR(tPlantCom_E2E_Out_10ms.analogSignals), ADR(tPlantCom_E2E_Out_Bus.analogSignals[iAnaArrayMax100ms+1]), (iAnaArrayMax10ms+1) * SIZEOF(tPlantCom_E2E_Out_10ms.analogSignals[0]));

	(*** Output to Masters  ***)
	FOR x:=iMasNumMin TO iMasNumMax DO
		memcpy(ADR(tPlantCom_E2M_Out_10ms[x].digitalSignals), ADR(tPlantCom_E2M_Out_Bus[x].digitalSignals[iDigArrayMax100ms+1]), (iDigArrayMax10ms+1) * SIZEOF(tPlantCom_E2M_Out_10ms[x].digitalSignals[0]));
		memcpy(ADR(tPlantCom_E2M_Out_10ms[x].analogSignals), ADR(tPlantCom_E2M_Out_Bus[x].analogSignals[iAnaArrayMax100ms+1]), (iAnaArrayMax10ms+1) * SIZEOF(tPlantCom_E2M_Out_10ms[x].analogSignals[0]));
	END_FOR;

END_PROGRAM
```

#### OutInit.st - Init code
```iecst
(*******************************************************************************
Mapping from Plc Arrays to Bus Arrays with force logic

This code is confidential and proprietary to the INNIO Company.
It may not be used in any form, or reproduced in any manner, without the express
written permission of the INNIO Company.
Copyright, INNIO Company, 2024

Customized modifications: -
------------------------

History:
-------
V4.14.0	26.11.2024	Astner	Created Task

Instructions for use: -
--------------------

Outstandings:
------------

*******************************************************************************)

PROGRAM _INIT
	(* Insert code here *)

END_PROGRAM
```

#### OutVariables.var - Local variables
```iecst
VAR
	idx : USINT := 0;
	x : USINT := 0;
END_VAR
```

### Program Logical/HalIO/PlantCommunication/xComMapOut100ms (IEC, version 4.14.0)

#### OutCyclic.st - Cyclic code
```iecst
(*******************************************************************************
Mapping from Plc Arrays to Bus Arrays with force logic

This code is confidential and proprietary to the INNIO Company.
It may not be used in any form, or reproduced in any manner, without the express
written permission of the INNIO Company.
Copyright, INNIO Company, 2024

Customized modifications: -
------------------------

History:
-------
V4.14.0	26.11.2024	Astner	Created Task

Instructions for use: -
--------------------

Outstandings:
------------

*******************************************************************************)
PROGRAM _CYCLIC
	(* Exit if configuration fails or not active *)
	IF (NOT MM2VIS.tPlantComm.bCfg_OK OR NOT Para.tPlantComm.bActive) THEN
		RETURN;
	END_IF;

	(***************************)
	(* Copy Data to Bus Arrays *)
	(***************************)

	(*** Output to Engines  ***)
	memcpy(ADR(tPlantCom_E2E_Out_Bus.digitalSignals), ADR(tPlantCom_E2E_Out_Plc.digitalSignals[0]), (iDigArrayMax100ms+1) * SIZEOF(tPlantCom_E2E_Out_Bus.digitalSignals[0]));
	memcpy(ADR(tPlantCom_E2E_Out_Bus.analogSignals), ADR(tPlantCom_E2E_Out_Plc.analogSignals[0]), (iAnaArrayMax100ms+1) * SIZEOF(tPlantCom_E2E_Out_Bus.analogSignals[0]));

	(*** Outputs to Masters  ***)
	FOR x:=iMasNumMin TO iMasNumMax DO
		memcpy(ADR(tPlantCom_E2M_Out_Bus[x].digitalSignals), ADR(tPlantCom_E2M_Out_Plc[x].digitalSignals[0]), (iDigArrayMax100ms+1) * SIZEOF(tPlantCom_E2M_Out_Bus[x].digitalSignals[0]));
		memcpy(ADR(tPlantCom_E2M_Out_Bus[x].analogSignals), ADR(tPlantCom_E2M_Out_Plc[x].analogSignals[0]), (iAnaArrayMax100ms+1) * SIZEOF(tPlantCom_E2M_Out_Bus[x].analogSignals[0]));
	END_FOR

	(************************************************)
	(* Overwrite forced outputs with value from HMI *)
	(************************************************)

	IF (MM2VIS.tPlantComm.iFrc_Gbl > 0) THEN
		IF (tPlantCom_E2E_Out_Hmi.iNum_ForcedValues > 0) THEN
			(* Digital Signals *)
			FOR idx:=0 TO iDigArrayMax100ms DO
				IF (tPlantCom_E2E_Out_Hmi.bDigForceActive[idx]) THEN
					tPlantCom_E2E_Out_Bus.digitalSignals[idx].Value := tPlantCom_E2E_Out_Hmi.bForceValue[idx];
					tPlantCom_E2E_Out_Bus.digitalSignals[idx].GoodQual := TRUE;
				END_IF
			END_FOR
			(* Analog Signals *)
			FOR idx:=0 TO iAnaArrayMax100ms DO
				IF (tPlantCom_E2E_Out_Hmi.bAnaForceActive[idx]) THEN
					tPlantCom_E2E_Out_Bus.analogSignals[idx].Value := tPlantCom_E2E_Out_Hmi.rForceValue[idx];
					tPlantCom_E2E_Out_Bus.analogSignals[idx].GoodQual := TRUE;
				END_IF
			END_FOR
		END_IF

		FOR x:=iMasNumMin TO iMasNumMax DO
			IF (tPlantCom_E2M_Out_Hmi[x].iNum_ForcedValues > 0) THEN
				(* Digital Signals *)
				FOR idx:=0 TO iDigArrayMax100ms DO
					IF (tPlantCom_E2M_Out_Hmi[x].bDigForceActive[idx]) THEN
						tPlantCom_E2M_Out_Bus[x].digitalSignals[idx].Value := tPlantCom_E2M_Out_Hmi[x].bForceValue[idx];
						tPlantCom_E2M_Out_Bus[x].digitalSignals[idx].GoodQual := TRUE;
					END_IF
				END_FOR
				(* Analog Signals *)
				FOR idx:=0 TO iAnaArrayMax100ms DO
					IF (tPlantCom_E2M_Out_Hmi[x].bAnaForceActive[idx]) THEN
						tPlantCom_E2M_Out_Bus[x].analogSignals[idx].Value := tPlantCom_E2M_Out_Hmi[x].rForceValue[idx];
						tPlantCom_E2M_Out_Bus[x].analogSignals[idx].GoodQual := TRUE;
					END_IF
				END_FOR
			END_IF
		END_FOR
	END_IF

	(*****************************************)
	(* Split Data into 100ms and 10ms Arrays *)
	(*****************************************)

	(*** Output to Engines  ***)
	(* Slow Signals *)
	memcpy(ADR(tPlantCom_E2E_Out_100ms.digitalSignals), ADR(tPlantCom_E2E_Out_Bus.digitalSignals[0]), (iDigArrayMax100ms+1) * SIZEOF(tPlantCom_E2E_Out_100ms.digitalSignals[0]));
	memcpy(ADR(tPlantCom_E2E_Out_100ms.analogSignals), ADR(tPlantCom_E2E_Out_Bus.analogSignals[0]), (iAnaArrayMax100ms+1) * SIZEOF(tPlantCom_E2E_Out_100ms.analogSignals[0]));

	(*** Output to Masters  ***)
	FOR x:=iMasNumMin TO iMasNumMax DO
		(* Slow Signals *)
		memcpy(ADR(tPlantCom_E2M_Out_100ms[x].digitalSignals), ADR(tPlantCom_E2M_Out_Bus[x].digitalSignals[0]), (iDigArrayMax100ms+1) * SIZEOF(tPlantCom_E2E_Out_100ms.digitalSignals[0]));
		memcpy(ADR(tPlantCom_E2M_Out_100ms[x].analogSignals), ADR(tPlantCom_E2M_Out_Bus[x].analogSignals[0]), (iAnaArrayMax100ms+1) * SIZEOF(tPlantCom_E2E_Out_100ms.analogSignals[0]));
	END_FOR
END_PROGRAM
```

#### OutInit.st - Init code
```iecst
(*******************************************************************************
Mapping from Plc Arrays to Bus Arrays with force logic

This code is confidential and proprietary to the INNIO Company.
It may not be used in any form, or reproduced in any manner, without the express
written permission of the INNIO Company.
Copyright, INNIO Company, 2024

Customized modifications: -
------------------------

History:
-------
V4.14.0	26.11.2024	Astner	Created Task

Instructions for use: -
--------------------

Outstandings:
------------

*******************************************************************************)

PROGRAM _INIT
	(* Insert code here *)

END_PROGRAM
```

#### OutVariables.var - Local variables
```iecst
VAR
	idx : USINT := 0;
	x : USINT := 0;
END_VAR
```

### Program Logical/HalIO/PlantCommunication/xComIO10ms (IEC, version 4.14.0)
